C03576=1024.617,175.946,-114.492,168.623,47.960,159.009
C03577=1024.611,175.697,-114.469,168.619,47.965,159.010
C03578=1024.606,175.448,-114.447,168.616,47.970,159.010
C03579=1024.600,175.200,-114.424,168.612,47.974,159.011
C03580=1024.594,174.951,-114.401,168.609,47.979,159.011
C03581=1024.589,174.701,-114.379,168.605,47.983,159.011
C03582=1024.583,174.452,-114.356,168.602,47.988,159.012
C03583=1024.577,174.203,-114.335,168.598,47.993,159.012
C03584=1024.572,173.955,-114.312,168.594,47.997,159.013
C03585=1024.566,173.706,-114.289,168.591,48.002,159.013
C03586=1024.560,173.457,-114.268,168.587,48.006,159.014
C03587=1024.554,173.208,-114.245,168.584,48.011,159.014
C03588=1024.548,172.959,-114.222,168.580,48.016,159.015
C03589=1024.543,172.710,-114.200,168.576,48.020,159.015
C03590=1024.537,172.461,-114.178,168.573,48.025,159.015
C03591=1024.531,172.178,-114.152,168.570,48.030,159.016
C03592=1024.525,171.896,-114.126,168.565,48.035,159.016
C03593=1024.518,171.612,-114.102,168.562,48.040,159.017
C03594=1024.512,171.330,-114.076,168.558,48.046,159.018
C03595=1024.506,171.080,-114.054,168.554,48.051,159.018
C03596=1024.500,170.832,-114.031,168.550,48.055,159.018
C03597=1024.495,170.583,-114.010,168.547,48.059,159.019
C03598=1024.489,170.334,-113.987,168.544,48.064,159.019
C03599=1024.483,170.085,-113.965,168.541,48.069,159.020
C03600=1024.477,169.836,-113.942,168.537,48.073,159.020
C03601=1024.472,169.587,-113.920,168.534,48.078,159.021
C03602=1024.466,169.338,-113.899,168.530,48.082,159.021
C03603=1024.461,169.089,-113.876,168.527,48.087,159.022
C03604=1024.456,168.840,-113.854,168.523,48.091,159.022
C03605=1024.450,168.591,-113.831,168.519,48.096,159.022
C03606=1024.444,168.342,-113.809,168.517,48.101,159.023
C03607=1024.439,168.093,-113.787,168.513,48.105,159.023
C03608=1024.433,167.844,-113.764,168.510,48.110,159.024
C03609=1024.427,167.595,-113.743,168.506,48.114,159.024
C03610=1024.422,167.347,-113.720,168.503,48.119,159.025
C03611=1024.417,167.097,-113.698,168.499,48.124,159.025
C03612=1024.410,166.848,-113.676,168.497,48.128,159.026
C03613=1024.405,166.600,-113.654,168.493,48.132,159.026
C03614=1024.400,166.350,-113.631,168.489,48.137,159.026
C03615=1024.394,166.101,-113.610,168.486,48.142,159.027
C03616=1024.389,165.853,-113.587,168.483,48.147,159.027
C03617=1024.383,165.604,-113.565,168.479,48.152,159.028
C03618=1024.378,165.355,-113.544,168.476,48.155,159.028
C03619=1024.372,165.106,-113.522,168.473,48.160,159.029
C03620=1024.366,164.857,-113.499,168.469,48.165,159.029
C03621=1024.361,164.608,-113.477,168.466,48.170,159.030
C03622=1024.355,164.359,-113.455,168.462,48.174,159.030
C03623=1024.350,164.110,-113.433,168.460,48.178,159.031
C03624=1024.344,163.861,-113.411,168.456,48.183,159.031
C03625=1024.339,163.612,-113.389,168.453,48.188,159.032
C03626=1024.334,163.363,-113.367,168.449,48.192,159.032
C03627=1024.328,163.114,-113.345,168.446,48.197,159.032
C03628=1024.323,162.865,-113.323,168.443,48.201,159.033
C03629=1024.317,162.616,-113.300,168.439,48.206,159.033
C03630=1024.312,162.367,-113.279,168.436,48.211,159.034
C03631=1024.306,162.118,-113.257,168.433,48.215,159.034
C03632=1024.301,161.869,-113.235,168.430,48.220,159.035
C03633=1024.295,161.621,-113.213,168.426,48.224,159.035
C03634=1024.290,161.372,-113.191,168.423,48.229,159.036
C03635=1024.285,161.122,-113.169,168.420,48.233,159.036
C03636=1024.279,160.874,-113.147,168.417,48.238,159.037
C03637=1024.274,160.624,-113.125,168.413,48.243,159.037
C03638=1024.269,160.375,-113.103,168.410,48.247,159.037
C03639=1024.263,160.126,-113.082,168.407,48.251,159.038
C03640=1024.258,159.878,-113.059,168.403,48.256,159.038
C03641=1024.252,159.628,-113.037,168.400,48.261,159.039
C03642=1024.247,159.380,-113.015,168.397,48.265,159.039
C03643=1024.241,159.130,-112.993,168.394,48.270,159.040
C03644=1024.236,158.882,-112.972,168.391,48.275,159.040
C03645=1024.229,158.633,-112.950,168.387,48.280,159.041
C03646=1024.225,158.383,-112.929,168.384,48.285,159.041
C03647=1024.219,158.134,-112.908,168.381,48.289,159.042
C03648=1024.213,157.886,-112.886,168.378,48.294,159.042
C03649=1024.207,157.636,-112.865,168.374,48.299,159.043
C03650=1024.202,157.388,-112.843,168.371,48.303,159.043
C03651=1024.196,157.138,-112.821,168.367,48.308,159.044
C03652=1024.190,156.890,-112.800,168.365,48.313,159.044
C03653=1024.185,156.640,-112.779,168.361,48.318,159.045
C03654=1024.179,156.392,-112.758,168.358,48.322,159.045
C03655=1024.173,156.108,-112.732,168.355,48.327,159.046
C03656=1024.166,155.825,-112.708,168.350,48.333,159.046
C03657=1024.160,155.541,-112.684,168.347,48.339,159.047
C03658=1024.153,155.258,-112.660,168.343,48.344,159.047
C03659=1024.148,155.010,-112.638,168.340,48.348,159.048
C03660=1024.142,154.760,-112.617,168.337,48.353,159.048
C03661=1024.137,154.511,-112.596,168.333,48.358,159.049
C03662=1024.131,154.262,-112.574,168.330,48.363,159.049
C03663=1024.125,154.013,-112.553,168.328,48.367,159.050
C03664=1024.119,153.764,-112.532,168.324,48.372,159.050
C03665=1024.114,153.515,-112.510,168.321,48.377,159.051
C03666=1024.109,153.266,-112.489,168.317,48.382,159.051
C03667=1024.103,153.016,-112.468,168.315,48.386,159.052
C03668=1024.098,152.768,-112.446,168.311,48.391,159.052
C03669=1024.091,152.519,-112.425,168.308,48.396,159.053
C03670=1024.086,152.270,-112.404,168.305,48.401,159.053
C03671=1024.080,152.020,-112.383,168.302,48.406,159.054
C03672=1024.074,151.772,-112.361,168.299,48.411,159.054
C03673=1024.069,151.523,-112.341,168.295,48.415,159.055
C03674=1024.063,151.274,-112.319,168.292,48.420,159.055
C03675=1024.058,151.024,-112.299,168.289,48.425,159.056
C03676=1024.052,150.775,-112.277,168.286,48.430,159.056
C03677=1024.046,150.527,-112.256,168.283,48.434,159.057
C03678=1024.041,150.278,-112.235,168.279,48.439,159.057
C03679=1024.035,150.028,-112.214,168.277,48.444,159.058
C03680=1024.029,149.779,-112.193,168.273,48.449,159.058
C03681=1024.024,149.531,-112.171,168.270,48.453,159.059
C03682=1024.019,149.281,-112.150,168.266,48.458,159.059
C03683=1024.013,149.032,-112.129,168.264,48.463,159.060
C03684=1024.008,148.783,-112.108,168.260,48.468,159.060
C03685=1024.002,148.534,-112.087,168.257,48.473,159.061
C03686=1023.996,148.285,-112.066,168.255,48.477,159.061
C03687=1023.991,148.036,-112.045,168.251,48.483,159.062
C03688=1023.985,147.786,-112.024,168.248,48.487,159.063
C03689=1023.979,147.538,-112.003,168.245,48.492,159.063
C03690=1023.974,147.289,-111.982,168.242,48.497,159.064
C03691=1023.967,147.040,-111.961,168.239,48.502,159.064
C03692=1023.962,146.791,-111.941,168.235,48.506,159.065
C03693=1023.957,146.542,-111.920,168.233,48.511,159.065
C03694=1023.951,146.292,-111.898,168.229,48.516,159.066
C03695=1023.945,146.043,-111.878,168.226,48.521,159.066
C03696=1023.940,145.795,-111.857,168.224,48.525,159.067
C03697=1023.934,145.545,-111.836,168.220,48.531,159.067
C03698=1023.929,145.296,-111.815,168.217,48.536,159.068
C03699=1023.922,145.048,-111.794,168.214,48.540,159.068
C03700=1023.917,144.799,-111.774,168.211,48.545,159.069
C03701=1023.911,144.549,-111.753,168.208,48.550,159.069
C03702=1023.906,144.300,-111.732,168.204,48.555,159.070
C03703=1023.900,144.051,-111.712,168.202,48.560,159.070
C03704=1023.894,143.802,-111.691,168.199,48.565,159.071
C03705=1023.889,143.552,-111.670,168.195,48.570,159.071
C03706=1023.883,143.303,-111.650,168.192,48.574,159.072
C03707=1023.878,143.055,-111.628,168.189,48.579,159.072
C03708=1023.871,142.805,-111.608,168.186,48.584,159.073
C03709=1023.866,142.556,-111.588,168.183,48.589,159.073
C03710=1023.861,142.307,-111.567,168.181,48.594,159.074
C03711=1023.855,142.059,-111.546,168.177,48.599,159.074
C03712=1023.848,141.809,-111.525,168.174,48.604,159.075
C03713=1023.843,141.560,-111.505,168.171,48.608,159.076
C03714=1023.838,141.311,-111.484,168.168,48.613,159.076
C03715=1023.833,141.062,-111.464,168.164,48.618,159.076
C03716=1023.826,140.813,-111.443,168.162,48.623,159.077
C03717=1023.821,140.564,-111.422,168.159,48.628,159.078
C03718=1023.815,140.315,-111.402,168.155,48.633,159.078
C03719=1023.809,140.031,-111.378,168.152,48.638,159.079
C03720=1023.802,139.748,-111.355,168.149,48.644,159.079
C03721=1023.796,139.463,-111.332,168.145,48.649,159.080
C03722=1023.790,139.180,-111.308,168.142,48.655,159.080
C03723=1023.785,138.931,-111.287,168.139,48.659,159.081
C03724=1023.779,138.682,-111.267,168.136,48.664,159.081
C03725=1023.773,138.433,-111.247,168.133,48.670,159.082
C03726=1023.768,138.184,-111.226,168.130,48.674,159.083
C03727=1023.762,137.934,-111.205,168.127,48.679,159.083
C03728=1023.756,137.686,-111.185,168.123,48.684,159.084
C03729=1023.751,137.437,-111.164,168.121,48.688,159.084
C03730=1023.745,137.188,-111.144,168.118,48.694,159.085
C03731=1023.739,136.939,-111.124,168.115,48.699,159.085
C03732=1023.733,136.690,-111.104,168.112,48.703,159.086
C03733=1023.728,136.440,-111.083,168.109,48.708,159.086
C03734=1023.723,136.190,-111.063,168.106,48.714,159.087
C03735=1023.717,135.942,-111.043,168.103,48.718,159.087
C03736=1023.711,135.693,-111.022,168.100,48.723,159.088
C03737=1023.705,135.444,-111.002,168.096,48.728,159.088
C03738=1023.700,135.195,-110.982,168.094,48.733,159.089
C03739=1023.694,134.946,-110.962,168.091,48.738,159.090
C03740=1023.688,134.696,-110.941,168.087,48.743,159.090
C03741=1023.682,134.447,-110.921,168.085,48.748,159.091
C03742=1023.677,134.198,-110.901,168.082,48.753,159.091
C03743=1023.671,133.949,-110.881,168.079,48.758,159.092
C03744=1023.666,133.700,-110.860,168.076,48.763,159.092
C03745=1023.660,133.451,-110.841,168.073,48.768,159.093
C03746=1023.655,133.202,-110.820,168.070,48.772,159.093
C03747=1023.649,132.953,-110.800,168.067,48.778,159.094
C03748=1023.644,132.704,-110.780,168.064,48.783,159.094
C03749=1023.638,132.455,-110.760,168.061,48.787,159.095
C03750=1023.632,132.205,-110.739,168.058,48.792,159.095
C03751=1023.626,131.956,-110.719,168.055,48.797,159.096
C03752=1023.621,131.706,-110.699,168.053,48.802,159.097
C03753=1023.615,131.458,-110.679,168.049,48.807,159.097
C03754=1023.609,131.208,-110.659,168.047,48.812,159.098
C03755=1023.603,130.960,-110.639,168.043,48.817,159.098
C03756=1023.598,130.711,-110.618,168.040,48.822,159.099
C03757=1023.593,130.461,-110.599,168.038,48.827,159.099
C03758=1023.587,130.212,-110.579,168.034,48.832,159.100
C03759=1023.581,129.963,-110.558,168.032,48.836,159.100
C03760=1023.576,129.714,-110.539,168.029,48.842,159.101
C03761=1023.570,129.465,-110.519,168.026,48.847,159.101
C03762=1023.564,129.216,-110.499,168.023,48.851,159.102
C03763=1023.558,128.967,-110.480,168.020,48.857,159.103
C03764=1023.553,128.718,-110.459,168.017,48.862,159.103
C03765=1023.547,128.468,-110.440,168.015,48.867,159.104
C03766=1023.540,128.219,-110.420,168.011,48.872,159.104
C03767=1023.534,127.970,-110.400,168.008,48.877,159.105
C03768=1023.529,127.720,-110.381,168.006,48.882,159.105
C03769=1023.523,127.472,-110.361,168.002,48.887,159.106
C03770=1023.517,127.222,-110.341,167.999,48.892,159.106
C03771=1023.512,126.973,-110.321,167.997,48.897,159.107
C03772=1023.506,126.724,-110.302,167.994,48.902,159.108
C03773=1023.500,126.475,-110.282,167.990,48.908,159.108
C03774=1023.494,126.225,-110.262,167.988,48.912,159.109
C03775=1023.488,125.976,-110.242,167.985,48.917,159.109
C03776=1023.483,125.727,-110.223,167.982,48.923,159.110
C03777=1023.477,125.478,-110.203,167.979,48.927,159.110
C03778=1023.471,125.229,-110.183,167.976,48.932,159.111
C03779=1023.466,124.980,-110.163,167.974,48.938,159.112
C03780=1023.460,124.730,-110.144,167.970,48.942,159.112
C03781=1023.454,124.481,-110.124,167.967,48.947,159.113
C03782=1023.448,124.232,-110.105,167.965,48.953,159.113
C03783=1023.442,123.948,-110.083,167.961,48.958,159.114
C03784=1023.435,123.665,-110.060,167.958,48.964,159.114
C03785=1023.429,123.381,-110.038,167.955,48.970,159.115
C03786=1023.422,123.097,-110.016,167.952,48.975,159.116
C03787=1023.418,122.849,-109.995,167.948,48.980,159.116
C03788=1023.412,122.600,-109.976,167.946,48.985,159.117
C03789=1023.406,122.351,-109.956,167.943,48.990,159.117
C03790=1023.400,122.101,-109.937,167.939,48.995,159.118
C03791=1023.394,121.852,-109.917,167.937,49.001,159.119
C03792=1023.389,121.603,-109.898,167.934,49.005,159.119
C03793=1023.383,121.354,-109.879,167.932,49.010,159.120
C03794=1023.377,121.105,-109.859,167.928,49.015,159.120
C03795=1023.372,120.855,-109.839,167.926,49.020,159.121
C03796=1023.366,120.606,-109.820,167.923,49.025,159.121
C03797=1023.360,120.357,-109.800,167.919,49.030,159.122
C03798=1023.355,120.107,-109.780,167.917,49.035,159.122
C03799=1023.349,119.859,-109.761,167.914,49.040,159.123
C03800=1023.343,119.610,-109.741,167.912,49.045,159.123
C03801=1023.338,119.360,-109.722,167.909,49.051,159.124
C03802=1023.332,119.112,-109.702,167.906,49.055,159.125
C03803=1023.327,118.862,-109.682,167.903,49.060,159.125
C03804=1023.321,118.612,-109.663,167.900,49.065,159.126
C03805=1023.315,118.364,-109.643,167.897,49.070,159.126
C03806=1023.309,118.114,-109.624,167.894,49.075,159.127
C03807=1023.304,117.865,-109.605,167.892,49.080,159.127
C03808=1023.299,117.616,-109.586,167.888,49.085,159.128
C03809=1023.293,117.367,-109.566,167.886,49.090,159.128
C03810=1023.287,117.118,-109.547,167.883,49.095,159.129
C03811=1023.281,116.868,-109.527,167.881,49.100,159.130
C03812=1023.276,116.619,-109.507,167.877,49.104,159.130
C03813=1023.271,116.370,-109.488,167.875,49.110,159.131
C03814=1023.265,116.121,-109.469,167.872,49.115,159.131
C03815=1023.260,115.872,-109.450,167.869,49.119,159.132
C03816=1023.254,115.623,-109.430,167.866,49.124,159.132
C03817=1023.248,115.373,-109.410,167.864,49.130,159.133
C03818=1023.243,115.125,-109.391,167.861,49.135,159.133
C03819=1023.237,114.875,-109.372,167.858,49.139,159.134
C03820=1023.231,114.626,-109.353,167.855,49.144,159.134
C03821=1023.226,114.377,-109.332,167.853,49.149,159.135
C03822=1023.220,114.127,-109.313,167.849,49.154,159.136
C03823=1023.215,113.878,-109.294,167.847,49.159,159.136
C03824=1023.210,113.629,-109.275,167.844,49.164,159.137
C03825=1023.204,113.380,-109.256,167.841,49.168,159.137
C03826=1023.198,113.131,-109.236,167.838,49.174,159.138
C03827=1023.193,112.882,-109.217,167.836,49.179,159.138
C03828=1023.187,112.633,-109.198,167.833,49.184,159.139
C03829=1023.182,112.383,-109.178,167.830,49.188,159.139
C03830=1023.176,112.134,-109.159,167.827,49.194,159.140
C03831=1023.170,111.884,-109.140,167.825,49.199,159.140
C03832=1023.165,111.636,-109.121,167.821,49.203,159.141
C03833=1023.159,111.386,-109.102,167.819,49.209,159.142
C03834=1023.153,111.137,-109.083,167.816,49.214,159.142
C03835=1023.147,110.888,-109.064,167.814,49.219,159.143
C03836=1023.142,110.639,-109.045,167.811,49.224,159.143
C03837=1023.137,110.389,-109.026,167.808,49.229,159.144
C03838=1023.131,110.140,-109.007,167.805,49.234,159.144
C03839=1023.124,109.891,-108.988,167.802,49.239,159.145
C03840=1023.119,109.642,-108.969,167.800,49.244,159.145
C03841=1023.114,109.393,-108.950,167.797,49.249,159.146
C03842=1023.107,109.144,-108.931,167.794,49.254,159.147
C03843=1023.102,108.894,-108.912,167.791,49.260,159.147
C03844=1023.097,108.645,-108.894,167.789,49.264,159.148
C03845=1023.090,108.396,-108.875,167.785,49.269,159.148
C03846=1023.085,108.146,-108.856,167.783,49.275,159.149
C03847=1023.078,107.862,-108.834,167.779,49.281,159.150
C03848=1023.072,107.579,-108.813,167.776,49.286,159.150
C03849=1023.065,107.295,-108.791,167.773,49.292,159.151
C03850=1023.058,107.011,-108.770,167.770,49.298,159.151
C03851=1023.053,106.762,-108.751,167.767,49.303,159.152
C03852=1023.047,106.513,-108.733,167.765,49.308,159.153
C03853=1023.041,106.264,-108.714,167.762,49.313,159.153
C03854=1023.036,106.014,-108.694,167.760,49.318,159.154
C03855=1023.030,105.765,-108.677,167.756,49.323,159.154
C03856=1023.024,105.516,-108.657,167.754,49.328,159.155
C03857=1023.018,105.267,-108.639,167.751,49.333,159.155
C03858=1023.013,105.018,-108.620,167.749,49.339,159.156
C03859=1023.008,104.768,-108.601,167.746,49.344,159.157
C03860=1023.001,104.519,-108.583,167.743,49.348,159.157
C03861=1022.996,104.270,-108.564,167.740,49.354,159.158
C03862=1022.990,104.021,-108.545,167.738,49.359,159.158
C03863=1022.984,103.771,-108.527,167.734,49.364,159.159
C03864=1022.979,103.522,-108.508,167.731,49.369,159.159
C03865=1022.973,103.273,-108.489,167.729,49.374,159.160
C03866=1022.967,103.024,-108.470,167.726,49.379,159.160
C03867=1022.962,102.774,-108.452,167.724,49.384,159.161
C03868=1022.956,102.525,-108.433,167.721,49.389,159.162
C03869=1022.950,102.276,-108.414,167.718,49.394,159.162
C03870=1022.945,102.027,-108.395,167.716,49.399,159.163
C03871=1022.939,101.777,-108.377,167.713,49.404,159.163
C03872=1022.934,101.529,-108.358,167.710,49.409,159.164
C03873=1022.927,101.279,-108.340,167.707,49.414,159.165
C03874=1022.922,101.029,-108.321,167.705,49.419,159.165
C03875=1022.917,100.781,-108.302,167.702,49.424,159.166
C03876=1022.910,100.532,-108.283,167.700,49.429,159.166
C03877=1022.906,100.282,-108.265,167.696,49.434,159.167
C03878=1022.900,100.033,-108.246,167.694,49.439,159.167
C03879=1022.894,99.783,-108.228,167.691,49.445,159.168
C03880=1022.889,99.534,-108.209,167.689,49.449,159.168
C03881=1022.882,99.285,-108.191,167.685,49.454,159.169
C03882=1022.877,99.035,-108.172,167.683,49.460,159.170
C03883=1022.871,98.787,-108.154,167.680,49.465,159.170
C03884=1022.865,98.537,-108.136,167.678,49.470,159.171
C03885=1022.860,98.288,-108.117,167.675,49.475,159.171
C03886=1022.854,98.039,-108.099,167.673,49.480,159.172
C03887=1022.847,97.789,-108.080,167.669,49.485,159.172
C03888=1022.843,97.540,-108.062,167.666,49.490,159.173
C03889=1022.836,97.291,-108.044,167.664,49.496,159.174
C03890=1022.831,97.042,-108.026,167.661,49.501,159.174
C03891=1022.825,96.792,-108.008,167.659,49.506,159.175
C03892=1022.819,96.543,-107.989,167.655,49.511,159.175
C03893=1022.813,96.294,-107.971,167.653,49.516,159.176
C03894=1022.808,96.044,-107.952,167.650,49.521,159.176
C03895=1022.802,95.795,-107.934,167.648,49.526,159.177
C03896=1022.796,95.546,-107.916,167.645,49.532,159.178
C03897=1022.791,95.297,-107.898,167.642,49.536,159.178
C03898=1022.785,95.047,-107.880,167.639,49.542,159.179
C03899=1022.779,94.799,-107.861,167.637,49.547,159.179
C03900=1022.774,94.548,-107.843,167.634,49.552,159.180
C03901=1022.768,94.300,-107.825,167.632,49.557,159.181
C03902=1022.762,94.050,-107.807,167.628,49.562,159.181
C03903=1022.756,93.801,-107.789,167.626,49.567,159.182
C03904=1022.750,93.552,-107.770,167.623,49.572,159.182
C03905=1022.745,93.303,-107.752,167.621,49.577,159.183
C03906=1022.739,93.053,-107.734,167.618,49.583,159.183
C03907=1022.734,92.804,-107.716,167.616,49.587,159.184
C03908=1022.728,92.555,-107.698,167.612,49.592,159.184
C03909=1022.722,92.306,-107.679,167.610,49.598,159.185
C03910=1022.716,92.056,-107.661,167.607,49.603,159.185
C03911=1022.710,91.773,-107.640,167.604,49.608,159.186
C03912=1022.703,91.488,-107.620,167.601,49.614,159.187
C03913=1022.697,91.205,-107.599,167.598,49.620,159.187
C03914=1022.691,90.922,-107.579,167.595,49.625,159.188
C03915=1022.684,90.672,-107.561,167.593,49.631,159.189
C03916=1022.679,90.423,-107.542,167.590,49.636,159.189
C03917=1022.673,90.174,-107.524,167.587,49.640,159.190
C03918=1022.668,89.925,-107.506,167.584,49.646,159.190
C03919=1022.662,89.674,-107.488,167.582,49.651,159.191
C03920=1022.657,89.426,-107.469,167.579,49.656,159.191
C03921=1022.651,89.177,-107.452,167.577,49.661,159.192
C03922=1022.645,88.927,-107.434,167.573,49.666,159.193
C03923=1022.639,88.678,-107.416,167.571,49.672,159.193
C03924=1022.633,88.428,-107.398,167.568,49.677,159.194
C03925=1022.628,88.179,-107.381,167.566,49.682,159.194
C03926=1022.622,87.930,-107.363,167.563,49.687,159.195
C03927=1022.616,87.681,-107.345,167.561,49.692,159.196
C03928=1022.610,87.432,-107.327,167.558,49.697,159.196
C03929=1022.604,87.183,-107.309,167.555,49.702,159.197
C03930=1022.598,86.933,-107.291,167.552,49.708,159.197
C03931=1022.593,86.684,-107.274,167.550,49.712,159.198
C03932=1022.587,86.435,-107.256,167.547,49.718,159.198
C03933=1022.581,86.185,-107.238,167.545,49.723,159.199
C03934=1022.575,85.936,-107.221,167.542,49.728,159.200
C03935=1022.569,85.686,-107.203,167.539,49.733,159.200
C03936=1022.564,85.437,-107.185,167.536,49.739,159.201
C03937=1022.558,85.187,-107.167,167.534,49.744,159.201
C03938=1022.552,84.938,-107.150,167.531,49.749,159.202
C03939=1022.547,84.689,-107.132,167.529,49.754,159.202
C03940=1022.540,84.440,-107.114,167.526,49.759,159.203
C03941=1022.535,84.191,-107.097,167.524,49.764,159.204
C03942=1022.529,83.941,-107.079,167.520,49.769,159.204
C03943=1022.523,83.692,-107.061,167.518,49.774,159.205
C03944=1022.518,83.443,-107.043,167.515,49.780,159.205
C03945=1022.512,83.193,-107.026,167.513,49.784,159.206
C03946=1022.506,82.944,-107.008,167.510,49.790,159.206
C03947=1022.501,82.695,-106.990,167.508,49.795,159.207
C03948=1022.495,82.445,-106.972,167.504,49.800,159.207
C03949=1022.489,82.196,-106.955,167.502,49.805,159.208
C03950=1022.483,81.947,-106.937,167.499,49.810,159.209
C03951=1022.477,81.697,-106.919,167.497,49.816,159.209
C03952=1022.472,81.448,-106.902,167.494,49.821,159.210
C03953=1022.466,81.199,-106.884,167.491,49.825,159.210
C03954=1022.460,80.950,-106.866,167.489,49.831,159.211
C03955=1022.455,80.700,-106.849,167.486,49.836,159.211
C03956=1022.449,80.451,-106.831,167.484,49.841,159.212
C03957=1022.443,80.202,-106.813,167.481,49.846,159.213
C03958=1022.438,79.952,-106.796,167.479,49.851,159.213
C03959=1022.432,79.703,-106.779,167.475,49.856,159.214
C03960=1022.426,79.453,-106.761,167.473,49.861,159.214
C03961=1022.421,79.204,-106.743,167.470,49.866,159.215
C03962=1022.415,78.955,-106.726,167.468,49.871,159.215
C03963=1022.409,78.705,-106.708,167.465,49.877,159.216
C03964=1022.404,78.456,-106.690,167.463,49.882,159.216
C03965=1022.398,78.207,-106.673,167.460,49.886,159.217
C03966=1022.392,77.958,-106.655,167.457,49.891,159.217
C03967=1022.387,77.708,-106.638,167.455,49.897,159.218
C03968=1022.381,77.459,-106.620,167.452,49.902,159.219
C03969=1022.376,77.210,-106.603,167.449,49.906,159.219
C03970=1022.369,76.960,-106.585,167.446,49.912,159.220
C03971=1022.364,76.711,-106.569,167.444,49.917,159.220
C03972=1022.358,76.462,-106.551,167.441,49.923,159.221
C03973=1022.353,76.213,-106.533,167.439,49.927,159.222
C03974=1022.346,75.963,-106.516,167.436,49.932,159.222
C03975=1022.340,75.679,-106.496,167.433,49.939,159.223
C03976=1022.333,75.396,-106.476,167.430,49.945,159.223
C03977=1022.327,75.112,-106.457,167.427,49.950,159.224
C03978=1022.320,74.828,-106.438,167.424,49.956,159.225
C03979=1022.314,74.579,-106.420,167.421,49.962,159.225
C03980=1022.309,74.330,-106.403,167.419,49.966,159.226
C03981=1022.302,74.080,-106.386,167.417,49.971,159.226
C03982=1022.297,73.831,-106.368,167.414,49.977,159.227
C03983=1022.292,73.582,-106.351,167.411,49.982,159.228
C03984=1022.285,73.333,-106.334,167.409,49.987,159.228
C03985=1022.279,73.083,-106.316,167.406,49.992,159.229
C03986=1022.274,72.833,-106.300,167.403,49.997,159.229
C03987=1022.268,72.584,-106.282,167.401,50.003,159.230
C03988=1022.262,72.335,-106.266,167.398,50.008,159.230
C03989=1022.256,72.085,-106.248,167.395,50.012,159.231
C03990=1022.251,71.836,-106.230,167.393,50.018,159.231
C03991=1022.245,71.587,-106.214,167.390,50.023,159.232
C03992=1022.239,71.338,-106.197,167.387,50.028,159.232
C03993=1022.234,71.088,-106.180,167.385,50.033,159.233
C03994=1022.227,70.839,-106.162,167.382,50.038,159.234
C03995=1022.222,70.589,-106.145,167.380,50.044,159.234
C03996=1022.217,70.340,-106.128,167.377,50.049,159.235
C03997=1022.211,70.091,-106.112,167.374,50.053,159.235
C03998=1022.205,69.842,-106.094,167.372,50.059,159.236
C03999=1022.200,69.593,-106.077,167.369,50.064,159.236
C04000=1022.193,69.343,-106.060,167.367,50.069,159.237
C04001=1022.188,69.094,-106.042,167.364,50.074,159.238
C04002=1022.182,68.844,-106.025,167.362,50.079,159.238
C04003=1022.176,68.595,-106.008,167.358,50.084,159.239
C04004=1022.171,68.346,-105.992,167.356,50.090,159.239
C04005=1022.164,68.095,-105.975,167.353,50.095,159.240
C04006=1022.159,67.846,-105.957,167.351,50.099,159.240
C04007=1022.153,67.597,-105.941,167.348,50.105,159.241
C04008=1022.147,67.348,-105.924,167.346,50.110,159.242
C04009=1022.141,67.099,-105.907,167.343,50.116,159.242
C04010=1022.136,66.850,-105.890,167.340,50.120,159.243
C04011=1022.130,66.600,-105.874,167.337,50.125,159.243
C04012=1022.124,66.350,-105.856,167.335,50.131,159.244
C04013=1022.118,66.101,-105.839,167.332,50.136,159.244
C04014=1022.113,65.852,-105.823,167.330,50.141,159.245
C04015=1022.107,65.602,-105.806,167.327,50.146,159.245
C04016=1022.101,65.353,-105.789,167.325,50.151,159.246
C04017=1022.095,65.104,-105.772,167.323,50.157,159.247
C04018=1022.090,64.854,-105.756,167.319,50.162,159.247
C04019=1022.084,64.605,-105.739,167.317,50.166,159.248
C04020=1022.078,64.355,-105.721,167.314,50.172,159.248
C04021=1022.072,64.106,-105.705,167.312,50.177,159.249
C04022=1022.066,63.857,-105.688,167.309,50.182,159.249
C04023=1022.060,63.607,-105.671,167.307,50.187,159.250
C04024=1022.055,63.358,-105.654,167.303,50.193,159.250
C04025=1022.049,63.108,-105.638,167.301,50.197,159.251
C04026=1022.043,62.860,-105.621,167.298,50.203,159.252
C04027=1022.037,62.610,-105.605,167.296,50.208,159.252
C04028=1022.031,62.360,-105.588,167.293,50.214,159.253
C04029=1022.025,62.111,-105.571,167.291,50.218,159.253
C04030=1022.019,61.861,-105.555,167.288,50.224,159.254
C04031=1022.013,61.612,-105.539,167.285,50.229,159.254
C04032=1022.007,61.362,-105.523,167.283,50.235,159.255
C04033=1022.001,61.114,-105.506,167.280,50.240,159.256
C04034=1021.996,60.864,-105.489,167.278,50.245,159.256
C04035=1021.990,60.615,-105.473,167.274,50.250,159.257
C04036=1021.984,60.365,-105.456,167.273,50.256,159.257
C04037=1021.978,60.116,-105.440,167.269,50.261,159.258
C04038=1021.972,59.867,-105.424,167.267,50.266,159.259
C04039=1021.965,59.549,-105.403,167.264,50.273,159.259
C04040=1021.957,59.232,-105.382,167.260,50.280,159.260
C04041=1021.950,58.915,-105.362,167.257,50.287,159.261
C04042=1021.942,58.598,-105.340,167.254,50.293,159.262
C04043=1021.937,58.348,-105.323,167.251,50.298,159.262
C04044=1021.931,58.099,-105.307,167.248,50.304,159.263
C04045=1021.924,57.849,-105.290,167.246,50.309,159.263
C04046=1021.918,57.599,-105.274,167.242,50.314,159.264
C04047=1021.912,57.350,-105.258,167.241,50.319,159.264
C04048=1021.906,57.101,-105.242,167.237,50.324,159.265
C04049=1021.900,56.851,-105.225,167.235,50.330,159.265
C04050=1021.895,56.602,-105.209,167.232,50.335,159.266
C04051=1021.889,56.352,-105.192,167.230,50.340,159.266
C04052=1021.883,56.103,-105.176,167.227,50.345,159.267
C04053=1021.877,55.854,-105.160,167.225,50.350,159.268
C04054=1021.871,55.604,-105.144,167.222,50.356,159.268
C04055=1021.865,55.355,-105.127,167.220,50.361,159.269
C04056=1021.859,55.106,-105.111,167.216,50.366,159.269
C04057=1021.854,54.856,-105.094,167.215,50.371,159.270
C04058=1021.848,54.607,-105.078,167.211,50.376,159.270
C04059=1021.843,54.358,-105.062,167.209,50.381,159.271
C04060=1021.837,54.109,-105.046,167.206,50.387,159.271
C04061=1021.831,53.859,-105.030,167.204,50.392,159.272
C04062=1021.825,53.609,-105.014,167.201,50.397,159.273
C04063=1021.819,53.360,-104.998,167.199,50.402,159.273
C04064=1021.813,53.111,-104.981,167.196,50.407,159.274
C04065=1021.808,52.861,-104.965,167.194,50.413,159.274
C04066=1021.802,52.612,-104.948,167.190,50.418,159.275
C04067=1021.796,52.362,-104.932,167.188,50.423,159.275
C04068=1021.790,52.113,-104.916,167.185,50.428,159.276
C04069=1021.784,51.864,-104.900,167.183,50.433,159.276
C04070=1021.778,51.614,-104.883,167.180,50.438,159.277
C04071=1021.774,51.381,-104.868,167.178,50.443,159.277
C04072=1021.768,51.149,-104.853,167.175,50.448,159.278
C04073=1021.763,50.916,-104.838,167.173,50.453,159.278
C04074=1021.757,50.684,-104.823,167.171,50.457,159.279
C04075=1021.752,50.450,-104.808,167.169,50.462,159.280
C04076=1021.747,50.218,-104.793,167.165,50.467,159.280
C04077=1021.742,49.985,-104.778,167.163,50.472,159.280
C04078=1021.736,49.752,-104.763,167.161,50.476,159.281
C04079=1021.730,49.503,-104.747,167.159,50.482,159.282
C04080=1021.725,49.254,-104.731,167.155,50.487,159.282
C04081=1021.719,49.005,-104.714,167.153,50.492,159.283
C04082=1021.713,48.756,-104.698,167.150,50.497,159.283
C04083=1021.708,48.505,-104.682,167.148,50.502,159.284
C04084=1021.702,48.256,-104.666,167.145,50.507,159.284
C04085=1021.696,48.007,-104.650,167.143,50.512,159.285
C04086=1021.690,47.757,-104.633,167.140,50.517,159.285
C04087=1021.684,47.509,-104.617,167.137,50.523,159.286
C04088=1021.679,47.259,-104.602,167.135,50.527,159.286
C04089=1021.673,47.009,-104.586,167.132,50.533,159.287
C04090=1021.667,46.760,-104.569,167.130,50.537,159.287
C04091=1021.661,46.511,-104.553,167.127,50.542,159.288
C04092=1021.656,46.260,-104.537,167.125,50.548,159.288
C04093=1021.651,46.012,-104.521,167.122,50.553,159.289
C04094=1021.645,45.762,-104.505,167.119,50.558,159.289
C04095=1021.639,45.513,-104.489,167.117,50.563,159.290
C04096=1021.633,45.263,-104.473,167.114,50.568,159.290
C04097=1021.627,45.014,-104.457,167.112,50.572,159.291
C04098=1021.622,44.765,-104.441,167.109,50.578,159.292
C04099=1021.616,44.516,-104.425,167.106,50.583,159.292
C04100=1021.610,44.266,-104.409,167.104,50.588,159.293
C04101=1021.604,44.016,-104.393,167.101,50.593,159.293
C04102=1021.599,43.767,-104.376,167.099,50.598,159.294
C04103=1021.593,43.483,-104.359,167.096,50.604,159.294
C04104=1021.586,43.199,-104.340,167.093,50.609,159.295
C04105=1021.580,42.914,-104.322,167.090,50.615,159.295
C04106=1021.574,42.631,-104.304,167.087,50.620,159.296
C04107=1021.568,42.382,-104.287,167.084,50.626,159.296
C04108=1021.562,42.132,-104.272,167.082,50.631,159.297
C04109=1021.556,41.883,-104.256,167.079,50.636,159.297
C04110=1021.551,41.633,-104.241,167.076,50.641,159.298
C04111=1021.545,41.384,-104.225,167.074,50.647,159.299
C04112=1021.539,41.134,-104.209,167.071,50.652,159.299
C04113=1021.532,40.885,-104.193,167.068,50.657,159.299
C04114=1021.527,40.636,-104.178,167.066,50.661,159.300
C04115=1021.521,40.386,-104.162,167.063,50.667,159.301
C04116=1021.516,40.136,-104.146,167.061,50.672,159.301
C04117=1021.510,39.887,-104.130,167.058,50.677,159.302
C04118=1021.505,39.638,-104.115,167.055,50.682,159.302
C04119=1021.498,39.388,-104.100,167.052,50.688,159.303
C04120=1021.492,39.139,-104.084,167.050,50.693,159.303
C04121=1021.487,38.889,-104.068,167.047,50.698,159.304
C04122=1021.481,38.640,-104.052,167.045,50.703,159.304
C04123=1021.476,38.390,-104.037,167.042,50.708,159.305
C04124=1021.469,38.141,-104.021,167.040,50.713,159.305
C04125=1021.463,37.891,-104.006,167.038,50.718,159.306
C04126=1021.458,37.643,-103.990,167.034,50.723,159.306
C04127=1021.452,37.393,-103.974,167.032,50.728,159.307
C04128=1021.447,37.143,-103.959,167.029,50.733,159.307
C04129=1021.441,36.894,-103.943,167.027,50.739,159.308
C04130=1021.435,36.644,-103.928,167.024,50.744,159.308
C04131=1021.429,36.394,-103.912,167.022,50.749,159.309
C04132=1021.423,36.145,-103.897,167.018,50.754,159.309
C04133=1021.418,35.896,-103.881,167.017,50.759,159.310
C04134=1021.412,35.646,-103.866,167.013,50.764,159.311
C04135=1021.406,35.396,-103.851,167.011,50.769,159.311
C04136=1021.400,35.148,-103.835,167.008,50.775,159.312
C04137=1021.394,34.898,-103.820,167.006,50.780,159.312
C04138=1021.388,34.648,-103.805,167.003,50.785,159.313
C04139=1021.382,34.399,-103.790,167.000,50.790,159.313
C04140=1021.376,34.150,-103.774,166.998,50.796,159.314
C04141=1021.371,33.900,-103.758,166.995,50.801,159.314
C04142=1021.365,33.651,-103.744,166.992,50.806,159.315
C04143=1021.359,33.401,-103.728,166.990,50.811,159.315
C04144=1021.353,33.152,-103.712,166.987,50.816,159.316
C04145=1021.348,32.903,-103.697,166.984,50.821,159.316
C04146=1021.341,32.653,-103.682,166.982,50.826,159.317
C04147=1021.336,32.403,-103.667,166.979,50.831,159.317
C04148=1021.330,32.154,-103.652,166.977,50.837,159.318
C04149=1021.324,31.904,-103.637,166.974,50.842,159.318
C04150=1021.318,31.655,-103.620,166.972,50.847,159.319
C04151=1021.312,31.406,-103.606,166.968,50.852,159.319
C04152=1021.307,31.156,-103.590,166.966,50.858,159.320
C04153=1021.301,30.907,-103.576,166.963,50.863,159.320
C04154=1021.295,30.657,-103.560,166.961,50.867,159.321
C04155=1021.289,30.407,-103.545,166.958,50.873,159.321
C04156=1021.284,30.159,-103.529,166.956,50.877,159.322
C04157=1021.277,29.909,-103.514,166.953,50.883,159.323
C04158=1021.272,29.660,-103.499,166.951,50.888,159.323
C04159=1021.267,29.410,-103.484,166.947,50.893,159.324
C04160=1021.260,29.160,-103.469,166.945,50.898,159.324
C04161=1021.255,28.911,-103.454,166.942,50.903,159.324
C04162=1021.249,28.661,-103.439,166.940,50.908,159.325
C04163=1021.244,28.412,-103.423,166.937,50.913,159.325
C04164=1021.237,28.162,-103.408,166.935,50.919,159.326
C04165=1021.232,27.912,-103.393,166.932,50.924,159.327
C04166=1021.226,27.663,-103.378,166.929,50.929,159.327
C04167=1021.219,27.379,-103.361,166.927,50.935,159.328
C04168=1021.213,27.095,-103.344,166.924,50.941,159.328
C04169=1021.206,26.811,-103.327,166.920,50.947,159.329
C04170=1021.199,26.527,-103.310,166.917,50.953,159.329
C04171=1021.194,26.277,-103.295,166.915,50.957,159.330
C04172=1021.188,26.028,-103.280,166.912,50.963,159.330
C04173=1021.182,25.779,-103.265,166.909,50.967,159.331
C04174=1021.176,25.529,-103.250,166.906,50.973,159.331
C04175=1021.170,25.279,-103.235,166.904,50.978,159.332
C04176=1021.164,25.030,-103.220,166.901,50.983,159.332
C04177=1021.159,24.780,-103.205,166.899,50.988,159.333
C04178=1021.153,24.531,-103.190,166.896,50.993,159.333
C04179=1021.147,24.282,-103.175,166.893,50.999,159.334
C04180=1021.141,24.032,-103.160,166.891,51.004,159.335
C04181=1021.135,23.782,-103.146,166.888,51.009,159.335
C04182=1021.130,23.533,-103.131,166.885,51.014,159.335
C04183=1021.123,23.284,-103.116,166.882,51.019,159.336
C04184=1021.118,23.034,-103.101,166.881,51.025,159.337
C04185=1021.112,22.785,-103.086,166.877,51.030,159.337
C04186=1021.106,22.536,-103.071,166.875,51.035,159.338
C04187=1021.100,22.286,-103.056,166.872,51.040,159.338
C04188=1021.095,22.036,-103.042,166.870,51.045,159.339
C04189=1021.089,21.786,-103.027,166.867,51.050,159.339
C04190=1021.083,21.537,-103.012,166.864,51.055,159.339
C04191=1021.077,21.288,-102.997,166.862,51.061,159.340
C04192=1021.071,21.039,-102.982,166.859,51.065,159.341
C04193=1021.066,20.789,-102.968,166.856,51.071,159.341
C04194=1021.060,20.539,-102.953,166.854,51.076,159.342
C04195=1021.054,20.290,-102.938,166.851,51.081,159.342
C04196=1021.048,20.040,-102.923,166.849,51.086,159.342
C04197=1021.043,19.791,-102.908,166.845,51.091,159.343
C04198=1021.037,19.541,-102.894,166.843,51.096,159.343
C04199=1021.031,19.292,-102.879,166.840,51.101,159.344
C04200=1021.025,19.042,-102.864,166.837,51.107,159.344
C04201=1021.020,18.792,-102.850,166.835,51.111,159.345
C04202=1021.014,18.543,-102.835,166.832,51.117,159.345
C04203=1021.008,18.294,-102.820,166.830,51.122,159.346
C04204=1021.002,18.044,-102.807,166.827,51.127,159.346
C04205=1020.996,17.795,-102.792,166.825,51.132,159.347
C04206=1020.990,17.546,-102.777,166.822,51.137,159.347
C04207=1020.984,17.295,-102.763,166.819,51.142,159.348
C04208=1020.979,17.046,-102.748,166.816,51.147,159.348
C04209=1020.973,16.797,-102.733,166.814,51.152,159.349
C04210=1020.967,16.547,-102.719,166.811,51.158,159.349
C04211=1020.961,16.298,-102.704,166.808,51.163,159.350
C04212=1020.955,16.048,-102.689,166.805,51.168,159.350
C04213=1020.950,15.799,-102.675,166.803,51.173,159.351
C04214=1020.944,15.550,-102.661,166.801,51.178,159.351
C04215=1020.938,15.299,-102.646,166.797,51.183,159.352
C04216=1020.933,15.050,-102.631,166.795,51.188,159.352
C04217=1020.927,14.801,-102.618,166.792,51.194,159.353
C04218=1020.921,14.551,-102.603,166.790,51.198,159.353
C04219=1020.915,14.302,-102.588,166.787,51.204,159.354
C04220=1020.910,14.052,-102.574,166.784,51.208,159.354
C04221=1020.903,13.803,-102.559,166.781,51.214,159.355
C04222=1020.898,13.553,-102.545,166.779,51.219,159.355
C04223=1020.892,13.303,-102.530,166.776,51.224,159.356
C04224=1020.886,13.054,-102.517,166.773,51.230,159.356
C04225=1020.880,12.805,-102.502,166.771,51.234,159.357
C04226=1020.874,12.555,-102.488,166.768,51.240,159.357
C04227=1020.868,12.305,-102.474,166.766,51.245,159.358
C04228=1020.863,12.056,-102.459,166.763,51.250,159.358
C04229=1020.857,11.806,-102.445,166.760,51.256,159.359
C04230=1020.851,11.557,-102.431,166.757,51.261,159.359
C04231=1020.844,11.274,-102.415,166.755,51.266,159.360
C04232=1020.837,10.992,-102.399,166.751,51.273,159.360
C04233=1020.831,10.709,-102.383,166.748,51.279,159.361
C04234=1020.824,10.426,-102.367,166.745,51.284,159.361
C04235=1020.818,10.177,-102.353,166.742,51.290,159.362
C04236=1020.813,9.928,-102.339,166.740,51.295,159.362
C04237=1020.806,9.678,-102.325,166.737,51.300,159.363
C04238=1020.800,9.429,-102.311,166.734,51.305,159.363
C04239=1020.795,9.179,-102.297,166.731,51.310,159.364
C04240=1020.789,8.929,-102.282,166.729,51.316,159.364
C04241=1020.783,8.680,-102.268,166.727,51.321,159.365
C04242=1020.778,8.430,-102.254,166.723,51.326,159.365
C04243=1020.772,8.181,-102.240,166.720,51.331,159.366
C04244=1020.765,7.931,-102.226,166.718,51.336,159.366
C04245=1020.759,7.682,-102.212,166.715,51.341,159.367
C04246=1020.754,7.432,-102.198,166.713,51.346,159.367
C04247=1020.749,7.183,-102.184,166.710,51.351,159.368
C04248=1020.742,6.933,-102.169,166.707,51.356,159.368
C04249=1020.737,6.683,-102.155,166.705,51.362,159.369
C04250=1020.730,6.434,-102.142,166.701,51.367,159.369
C04251=1020.725,6.185,-102.128,166.699,51.372,159.370
C04252=1020.719,5.934,-102.114,166.696,51.377,159.370
C04253=1020.713,5.685,-102.099,166.694,51.382,159.371
C04254=1020.708,5.436,-102.086,166.691,51.387,159.371
C04255=1020.702,5.186,-102.072,166.688,51.393,159.371
C04256=1020.696,4.937,-102.058,166.685,51.398,159.372
C04257=1020.690,4.687,-102.043,166.682,51.403,159.372
C04258=1020.684,4.438,-102.030,166.680,51.408,159.373
C04259=1020.679,4.188,-102.016,166.677,51.413,159.373
C04260=1020.673,3.939,-102.002,166.675,51.418,159.374
C04261=1020.668,3.689,-101.988,166.672,51.423,159.374
C04262=1020.661,3.439,-101.974,166.670,51.428,159.375
C04263=1020.655,3.190,-101.960,166.666,51.433,159.375
C04264=1020.650,2.940,-101.946,166.663,51.438,159.375
C04265=1020.644,2.691,-101.932,166.661,51.443,159.376
C04266=1020.639,2.441,-101.918,166.658,51.448,159.376
C04267=1020.633,2.192,-101.904,166.656,51.453,159.377
C04268=1020.626,1.942,-101.891,166.653,51.458,159.377
C04269=1020.621,1.692,-101.877,166.650,51.463,159.378
C04270=1020.615,1.443,-101.863,166.647,51.469,159.378
C04271=1020.610,1.194,-101.848,166.645,51.473,159.379
C04272=1020.604,0.944,-101.835,166.642,51.479,159.379
C04273=1020.598,0.695,-101.821,166.639,51.484,159.380
C04274=1020.592,0.445,-101.807,166.637,51.489,159.380
C04275=1020.587,0.196,-101.794,166.634,51.494,159.380
C04276=1020.581,-0.055,-101.779,166.631,51.499,159.381
C04277=1020.575,-0.304,-101.765,166.628,51.504,159.381
C04278=1020.570,-0.554,-101.752,166.626,51.509,159.382
C04279=1020.564,-0.803,-101.738,166.623,51.514,159.382
C04280=1020.558,-1.053,-101.724,166.620,51.518,159.383
C04281=1020.553,-1.302,-101.711,166.617,51.524,159.383
C04282=1020.547,-1.552,-101.697,166.615,51.529,159.384
C04283=1020.542,-1.801,-101.683,166.612,51.534,159.384
C04284=1020.536,-2.051,-101.670,166.610,51.539,159.384
C04285=1020.530,-2.300,-101.656,166.607,51.544,159.385
C04286=1020.525,-2.550,-101.642,166.605,51.549,159.385
C04287=1020.519,-2.799,-101.628,166.601,51.553,159.386
C04288=1020.513,-3.050,-101.614,166.598,51.559,159.386
C04289=1020.507,-3.299,-101.601,166.596,51.564,159.387
C04290=1020.501,-3.548,-101.587,166.593,51.569,159.387
C04291=1020.496,-3.798,-101.573,166.590,51.574,159.387
C04292=1020.490,-4.048,-101.559,166.587,51.579,159.388
C04293=1020.485,-4.297,-101.545,166.585,51.584,159.388
C04294=1020.479,-4.546,-101.532,166.582,51.589,159.389
C04295=1020.473,-4.827,-101.517,166.579,51.594,159.389
C04296=1020.466,-5.108,-101.502,166.576,51.600,159.390
C04297=1020.459,-5.389,-101.487,166.573,51.606,159.390
C04298=1020.453,-5.670,-101.472,166.569,51.612,159.391
C04299=1020.447,-5.919,-101.459,166.567,51.617,159.391
C04300=1020.441,-6.168,-101.445,166.564,51.623,159.392
C04301=1020.435,-6.418,-101.432,166.561,51.628,159.392
C04302=1020.430,-6.668,-101.418,166.559,51.633,159.393
C04303=1020.423,-6.917,-101.405,166.556,51.638,159.393
C04304=1020.418,-7.167,-101.391,166.554,51.643,159.394
C04305=1020.412,-7.416,-101.378,166.551,51.648,159.394
C04306=1020.407,-7.666,-101.365,166.547,51.653,159.394
C04307=1020.400,-7.915,-101.352,166.545,51.658,159.395
C04308=1020.394,-8.165,-101.338,166.542,51.664,159.395
C04309=1020.389,-8.415,-101.325,166.539,51.669,159.396
C04310=1020.383,-8.664,-101.312,166.537,51.674,159.396
C04311=1020.377,-8.914,-101.298,166.533,51.678,159.396
C04312=1020.371,-9.164,-101.285,166.531,51.683,159.397
C04313=1020.366,-9.413,-101.272,166.528,51.688,159.397
C04314=1020.360,-9.662,-101.258,166.525,51.694,159.398
C04315=1020.355,-9.913,-101.245,166.523,51.699,159.398
C04316=1020.348,-10.162,-101.232,166.520,51.704,159.399
C04317=1020.342,-10.411,-101.219,166.517,51.709,159.399
C04318=1020.337,-10.661,-101.205,166.514,51.714,159.400
C04319=1020.331,-10.911,-101.192,166.511,51.719,159.400
C04320=1020.326,-11.160,-101.179,166.509,51.724,159.400
C04321=1020.320,-11.409,-101.166,166.506,51.730,159.401
C04322=1020.314,-11.659,-101.152,166.503,51.735,159.401
C04323=1020.309,-11.909,-101.140,166.501,51.740,159.402
C04324=1020.302,-12.158,-101.126,166.498,51.745,159.402
C04325=1020.297,-12.408,-101.113,166.495,51.749,159.402
C04326=1020.291,-12.658,-101.100,166.492,51.754,159.403
C04327=1020.285,-12.907,-101.086,166.489,51.760,159.403
C04328=1020.280,-13.157,-101.074,166.487,51.765,159.404
C04329=1020.274,-13.407,-101.060,166.484,51.770,159.404
C04330=1020.269,-13.656,-101.048,166.481,51.775,159.405
C04331=1020.263,-13.905,-101.034,166.478,51.780,159.405
C04332=1020.257,-14.155,-101.021,166.476,51.784,159.405
C04333=1020.251,-14.405,-101.008,166.473,51.790,159.406
C04334=1020.246,-14.655,-100.995,166.470,51.795,159.406
C04335=1020.240,-14.904,-100.981,166.467,51.800,159.407
C04336=1020.234,-15.154,-100.969,166.464,51.805,159.407
C04337=1020.229,-15.403,-100.955,166.462,51.809,159.407
C04338=1020.223,-15.653,-100.943,166.459,51.814,159.408
C04339=1020.218,-15.902,-100.929,166.456,51.820,159.408
C04340=1020.212,-16.152,-100.916,166.453,51.825,159.409
C04341=1020.206,-16.401,-100.903,166.450,51.830,159.409
C04342=1020.200,-16.651,-100.891,166.447,51.835,159.409
C04343=1020.194,-16.901,-100.878,166.445,51.840,159.410
C04344=1020.189,-17.150,-100.865,166.442,51.845,159.410
C04345=1020.183,-17.400,-100.852,166.439,51.851,159.411
C04346=1020.177,-17.650,-100.839,166.437,51.856,159.411
C04347=1020.171,-17.899,-100.826,166.434,51.861,159.412
C04348=1020.165,-18.149,-100.814,166.430,51.866,159.412
C04349=1020.160,-18.398,-100.801,166.428,51.871,159.413
C04350=1020.153,-18.647,-100.788,166.425,51.876,159.413
C04351=1020.148,-18.898,-100.775,166.422,51.881,159.413
C04352=1020.142,-19.147,-100.763,166.420,51.886,159.414
C04353=1020.136,-19.397,-100.750,166.416,51.891,159.414
C04354=1020.131,-19.646,-100.737,166.413,51.896,159.414
C04355=1020.125,-19.896,-100.724,166.411,51.901,159.415
C04356=1020.119,-20.146,-100.712,166.408,51.907,159.415
C04357=1020.113,-20.396,-100.699,166.406,51.912,159.416
C04358=1020.108,-20.644,-100.686,166.403,51.917,159.416
C04359=1020.101,-20.923,-100.672,166.400,51.922,159.417
C04360=1020.094,-21.203,-100.658,166.397,51.928,159.417
C04361=1020.089,-21.481,-100.644,166.393,51.934,159.418
C04362=1020.082,-21.761,-100.629,166.390,51.939,159.418
C04363=1020.077,-22.010,-100.617,166.388,51.944,159.418
C04364=1020.071,-22.259,-100.604,166.384,51.949,159.419
C04365=1020.065,-22.509,-100.591,166.381,51.955,159.419
C04366=1020.059,-22.758,-100.579,166.379,51.959,159.420
C04367=1020.053,-23.008,-100.566,166.376,51.965,159.420
C04368=1020.048,-23.258,-100.554,166.373,51.969,159.420
C04369=1020.042,-23.508,-100.541,166.371,51.974,159.421
C04370=1020.037,-23.757,-100.528,166.367,51.980,159.421
C04371=1020.031,-24.007,-100.515,166.364,51.985,159.422
C04372=1020.025,-24.257,-100.503,166.362,51.989,159.422
C04373=1020.020,-24.506,-100.491,166.359,51.994,159.422
C04374=1020.014,-24.756,-100.478,166.357,51.999,159.423
C04375=1020.008,-25.006,-100.465,166.353,52.005,159.423
C04376=1020.003,-25.255,-100.453,166.350,52.010,159.424
C04377=1019.997,-25.505,-100.440,166.348,52.014,159.424
C04378=1019.991,-25.755,-100.428,166.345,52.019,159.424
C04379=1019.986,-26.003,-100.415,166.343,52.024,159.425
C04380=1019.980,-26.253,-100.402,166.340,52.030,159.425
C04381=1019.974,-26.503,-100.390,166.336,52.034,159.425
C04382=1019.969,-26.752,-100.377,166.334,52.039,159.426
C04383=1019.963,-27.002,-100.365,166.331,52.045,159.426
C04384=1019.957,-27.252,-100.352,166.327,52.049,159.426
C04385=1019.952,-27.502,-100.339,166.325,52.054,159.427
C04386=1019.946,-27.752,-100.327,166.322,52.059,159.427
C04387=1019.940,-28.001,-100.315,166.320,52.064,159.428
C04388=1019.934,-28.250,-100.303,166.317,52.070,159.428
C04389=1019.929,-28.501,-100.291,166.314,52.075,159.429
C04390=1019.924,-28.750,-100.279,166.310,52.079,159.429
C04391=1019.918,-29.000,-100.266,166.308,52.084,159.429
C04392=1019.912,-29.250,-100.254,166.305,52.090,159.430
C04393=1019.906,-29.499,-100.241,166.302,52.095,159.430
C04394=1019.900,-29.748,-100.229,166.300,52.100,159.431
C04395=1019.895,-29.998,-100.217,166.297,52.105,159.431
C04396=1019.889,-30.248,-100.205,166.294,52.111,159.431
C04397=1019.883,-30.498,-100.193,166.291,52.115,159.432
C04398=1019.878,-30.747,-100.181,166.288,52.120,159.432
C04399=1019.872,-30.997,-100.168,166.285,52.125,159.432
C04400=1019.866,-31.246,-100.157,166.282,52.131,159.433
C04401=1019.860,-31.496,-100.144,166.280,52.136,159.433
C04402=1019.855,-31.745,-100.132,166.276,52.140,159.433
C04403=1019.849,-31.996,-100.120,166.273,52.146,159.434
C04404=1019.843,-32.245,-100.107,166.271,52.151,159.434
C04405=1019.838,-32.495,-100.095,166.268,52.156,159.435
C04406=1019.831,-32.744,-100.083,166.265,52.161,159.435
C04407=1019.826,-32.994,-100.072,166.262,52.165,159.435
C04408=1019.820,-33.244,-100.059,166.259,52.171,159.436
C04409=1019.815,-33.493,-100.047,166.256,52.176,159.436
C04410=1019.809,-33.743,-100.035,166.254,52.181,159.437
C04411=1019.804,-33.993,-100.023,166.251,52.186,159.437
C04412=1019.797,-34.242,-100.011,166.247,52.191,159.437
C04413=1019.792,-34.491,-99.999,166.245,52.196,159.438
C04414=1019.786,-34.741,-99.986,166.242,52.201,159.438
C04415=1019.781,-34.991,-99.975,166.239,52.206,159.438
C04416=1019.775,-35.241,-99.962,166.237,52.211,159.439
C04417=1019.770,-35.490,-99.950,166.234,52.216,159.439
C04418=1019.764,-35.740,-99.939,166.230,52.221,159.439
C04419=1019.758,-35.990,-99.927,166.228,52.226,159.440
C04420=1019.752,-36.239,-99.914,166.225,52.231,159.440
C04421=1019.747,-36.489,-99.902,166.221,52.236,159.440
C04422=1019.742,-36.738,-99.890,166.219,52.241,159.441
C04423=1019.735,-37.017,-99.877,166.216,52.246,159.441
C04424=1019.729,-37.294,-99.864,166.213,52.251,159.442
C04425=1019.723,-37.573,-99.851,166.209,52.258,159.442
C04426=1019.717,-37.850,-99.837,166.206,52.263,159.443
C04427=1019.711,-38.100,-99.825,166.204,52.267,159.443
C04428=1019.706,-38.350,-99.813,166.201,52.273,159.443
C04429=1019.700,-38.600,-99.801,166.198,52.278,159.444
C04430=1019.694,-38.849,-99.789,166.195,52.282,159.444
C04431=1019.688,-39.099,-99.777,166.192,52.287,159.444
C04432=1019.683,-39.349,-99.765,166.189,52.293,159.445
C04433=1019.677,-39.598,-99.754,166.186,52.297,159.445
C04434=1019.671,-39.848,-99.742,166.183,52.302,159.445
C04435=1019.666,-40.098,-99.730,166.180,52.308,159.446
C04436=1019.660,-40.347,-99.718,166.177,52.313,159.446
C04437=1019.655,-40.597,-99.707,166.175,52.318,159.447
C04438=1019.649,-40.847,-99.696,166.172,52.323,159.447
C04439=1019.643,-41.096,-99.683,166.168,52.328,159.447
C04440=1019.637,-41.346,-99.673,166.166,52.333,159.448
C04441=1019.631,-41.596,-99.660,166.163,52.338,159.448
C04442=1019.626,-41.845,-99.649,166.160,52.343,159.448
C04443=1019.621,-42.095,-99.638,166.157,52.348,159.449
C04444=1019.614,-42.345,-99.626,166.155,52.353,159.449
C04445=1019.609,-42.595,-99.614,166.152,52.359,159.449
C04446=1019.604,-42.844,-99.602,166.148,52.363,159.450
C04447=1019.597,-43.094,-99.591,166.146,52.368,159.450
C04448=1019.592,-43.344,-99.579,166.143,52.373,159.451
C04449=1019.586,-43.593,-99.568,166.139,52.378,159.451
C04450=1019.581,-43.843,-99.556,166.136,52.383,159.451
C04451=1019.575,-44.093,-99.545,166.134,52.388,159.452
C04452=1019.570,-44.342,-99.533,166.131,52.393,159.452
C04453=1019.564,-44.591,-99.522,166.128,52.398,159.452
C04454=1019.558,-44.842,-99.510,166.126,52.403,159.453
C04455=1019.552,-45.091,-99.499,166.122,52.408,159.453
C04456=1019.547,-45.340,-99.487,166.119,52.413,159.453
C04457=1019.541,-45.591,-99.476,166.117,52.418,159.454
C04458=1019.536,-45.840,-99.464,166.113,52.423,159.454
C04459=1019.531,-46.090,-99.452,166.110,52.428,159.454
C04460=1019.525,-46.339,-99.441,166.108,52.433,159.455
C04461=1019.519,-46.590,-99.429,166.105,52.438,159.455
C04462=1019.513,-46.838,-99.418,166.102,52.443,159.455
C04463=1019.508,-47.088,-99.406,166.100,52.448,159.456
C04464=1019.503,-47.338,-99.396,166.096,52.453,159.456
C04465=1019.497,-47.588,-99.384,166.093,52.458,159.456
C04466=1019.491,-47.838,-99.373,166.090,52.463,159.456
C04467=1019.486,-48.087,-99.361,166.088,52.468,159.457
C04468=1019.480,-48.336,-99.350,166.085,52.473,159.457
C04469=1019.475,-48.587,-99.338,166.081,52.478,159.457
C04470=1019.469,-48.836,-99.327,166.079,52.483,159.458
C04471=1019.464,-49.086,-99.316,166.075,52.487,159.458
C04472=1019.458,-49.335,-99.304,166.073,52.492,159.459
C04473=1019.453,-49.585,-99.292,166.070,52.497,159.459
C04474=1019.446,-49.835,-99.281,166.067,52.502,159.459
C04475=1019.441,-50.085,-99.270,166.064,52.507,159.459
C04476=1019.436,-50.334,-99.259,166.061,52.512,159.460
C04477=1019.431,-50.584,-99.247,166.058,52.517,159.460
C04478=1019.425,-50.833,-99.236,166.056,52.522,159.460
C04479=1019.420,-51.083,-99.224,166.053,52.527,159.461
C04480=1019.413,-51.333,-99.213,166.049,52.532,159.461
C04481=1019.408,-51.583,-99.203,166.046,52.537,159.461
C04482=1019.402,-51.833,-99.192,166.043,52.542,159.462
C04483=1019.396,-52.082,-99.181,166.041,52.547,159.462
C04484=1019.391,-52.332,-99.170,166.038,52.553,159.463
C04485=1019.385,-52.581,-99.159,166.034,52.557,159.463
C04486=1019.379,-52.832,-99.148,166.031,52.563,159.463
C04487=1019.373,-53.110,-99.136,166.029,52.569,159.464
C04488=1019.366,-53.387,-99.124,166.026,52.574,159.464
C04489=1019.360,-53.666,-99.111,166.021,52.580,159.464
C04490=1019.354,-53.944,-99.100,166.018,52.585,159.465
C04491=1019.348,-54.194,-99.089,166.015,52.591,159.465
C04492=1019.342,-54.443,-99.078,166.012,52.596,159.465
C04493=1019.337,-54.693,-99.066,166.010,52.601,159.466
C04494=1019.331,-54.943,-99.055,166.007,52.606,159.466
C04495=1019.325,-55.193,-99.045,166.004,52.611,159.466
///RCONF 1,0,0,1,0,0,0,0,0,0,0,0,0,0,0,0,0,0,0,0,0,0,0,0
C04496=1019.320,-55.443,-99.034,166.001,52.616,159.467
C04497=1019.314,-55.692,-99.023,165.997,52.621,159.467
C04498=1019.308,-55.942,-99.012,165.995,52.626,159.467
C04499=1019.302,-56.191,-99.001,165.992,52.631,159.468
C04500=1019.297,-56.442,-98.991,165.989,52.637,159.468
C04501=1019.291,-56.691,-98.980,165.985,52.641,159.468
C04502=1019.286,-56.941,-98.969,165.983,52.646,159.469
C04503=1019.281,-57.190,-98.958,165.980,52.652,159.469
C04504=1019.275,-57.440,-98.947,165.977,52.657,159.469
C04505=1019.269,-57.690,-98.937,165.974,52.662,159.470
C04506=1019.264,-57.939,-98.926,165.972,52.667,159.470
C04507=1019.258,-58.189,-98.915,165.968,52.672,159.470
C04508=1019.252,-58.438,-98.904,165.965,52.677,159.471
C04509=1019.247,-58.688,-98.894,165.962,52.682,159.471
C04510=1019.241,-58.938,-98.883,165.960,52.687,159.471
C04511=1019.235,-59.187,-98.872,165.957,52.692,159.472
C04512=1019.231,-59.438,-98.862,165.954,52.697,159.472
C04513=1019.225,-59.687,-98.851,165.950,52.702,159.472
C04514=1019.219,-59.937,-98.840,165.948,52.707,159.473
C04515=1019.213,-60.186,-98.829,165.945,52.712,159.473
C04516=1019.208,-60.436,-98.819,165.941,52.717,159.473
C04517=1019.202,-60.686,-98.808,165.938,52.722,159.474
C04518=1019.196,-60.935,-98.797,165.936,52.727,159.474
C04519=1019.191,-61.186,-98.787,165.933,52.732,159.474
C04520=1019.185,-61.435,-98.776,165.929,52.737,159.475
C04521=1019.180,-61.685,-98.766,165.926,52.742,159.475
C04522=1019.174,-61.935,-98.755,165.924,52.747,159.475
C04523=1019.168,-62.184,-98.744,165.921,52.752,159.476
C04524=1019.164,-62.435,-98.733,165.918,52.757,159.476
C04525=1019.158,-62.684,-98.723,165.914,52.762,159.476
C04526=1019.152,-62.934,-98.712,165.912,52.767,159.477
C04527=1019.147,-63.184,-98.701,165.909,52.772,159.477
C04528=1019.141,-63.433,-98.691,165.906,52.777,159.477
C04529=1019.136,-63.683,-98.680,165.903,52.782,159.477
C04530=1019.130,-63.933,-98.670,165.900,52.787,159.478
C04531=1019.125,-64.182,-98.660,165.897,52.792,159.478
C04532=1019.119,-64.432,-98.649,165.894,52.797,159.478
C04533=1019.113,-64.681,-98.638,165.892,52.802,159.479
C04534=1019.108,-64.931,-98.628,165.888,52.806,159.479
C04535=1019.102,-65.181,-98.617,165.885,52.812,159.479
C04536=1019.097,-65.431,-98.607,165.882,52.816,159.479
C04537=1019.091,-65.680,-98.596,165.880,52.822,159.480
C04538=1019.086,-65.931,-98.585,165.876,52.826,159.480
C04539=1019.081,-66.180,-98.575,165.873,52.832,159.480
C04540=1019.076,-66.430,-98.565,165.871,52.836,159.481
C04541=1019.070,-66.679,-98.554,165.868,52.841,159.481
C04542=1019.065,-66.929,-98.543,165.864,52.846,159.481
C04543=1019.059,-67.179,-98.533,165.861,52.851,159.482
C04544=1019.054,-67.429,-98.522,165.859,52.856,159.482
C04545=1019.049,-67.678,-98.513,165.856,52.861,159.482
C04546=1019.043,-67.928,-98.502,165.852,52.866,159.482
C04547=1019.038,-68.178,-98.492,165.850,52.871,159.483
C04548=1019.032,-68.427,-98.481,165.847,52.875,159.483
C04549=1019.026,-68.677,-98.471,165.843,52.880,159.483
C04550=1019.021,-68.926,-98.460,165.840,52.886,159.483
C04551=1019.016,-69.206,-98.449,165.837,52.891,159.484
C04552=1019.010,-69.486,-98.437,165.834,52.896,159.484
C04553=1019.003,-69.765,-98.425,165.831,52.902,159.485
C04554=1018.997,-70.045,-98.413,165.827,52.907,159.485
C04555=1018.992,-70.294,-98.404,165.824,52.912,159.485
C04556=1018.986,-70.544,-98.393,165.821,52.917,159.485
C04557=1018.981,-70.794,-98.382,165.818,52.922,159.485
C04558=1018.975,-71.044,-98.372,165.815,52.926,159.486
C04559=1018.970,-71.293,-98.362,165.812,52.932,159.486
C04560=1018.965,-71.543,-98.352,165.809,52.936,159.486
C04561=1018.959,-71.793,-98.341,165.807,52.941,159.487
C04562=1018.954,-72.043,-98.331,165.803,52.946,159.487
C04563=1018.950,-72.292,-98.320,165.800,52.951,159.487
C04564=1018.944,-72.542,-98.310,165.798,52.956,159.488
C04565=1018.938,-72.792,-98.299,165.794,52.960,159.488
C04566=1018.934,-73.041,-98.289,165.791,52.965,159.488
C04567=1018.928,-73.291,-98.279,165.789,52.970,159.488
C04568=1018.923,-73.541,-98.269,165.786,52.975,159.488
C04569=1018.918,-73.790,-98.259,165.782,52.980,159.489
C04570=1018.912,-74.040,-98.248,165.780,52.985,159.489
C04571=1018.907,-74.290,-98.238,165.777,52.989,159.489
C04572=1018.901,-74.541,-98.228,165.774,52.995,159.490
C04573=1018.896,-74.789,-98.218,165.770,52.999,159.490
C04574=1018.890,-75.039,-98.208,165.768,53.004,159.490
C04575=1018.884,-75.289,-98.198,165.765,53.009,159.490
C04576=1018.880,-75.539,-98.188,165.762,53.015,159.491
C04577=1018.873,-75.788,-98.178,165.758,53.019,159.491
C04578=1018.868,-76.039,-98.168,165.756,53.024,159.491
C04579=1018.863,-76.288,-98.158,165.753,53.030,159.492
C04580=1018.858,-76.538,-98.148,165.750,53.034,159.492
C04581=1018.852,-76.787,-98.139,165.747,53.040,159.492
C04582=1018.847,-77.037,-98.129,165.744,53.044,159.492
C04583=1018.841,-77.287,-98.119,165.741,53.050,159.493
C04584=1018.837,-77.537,-98.109,165.738,53.054,159.493
C04585=1018.830,-77.787,-98.099,165.735,53.060,159.493
C04586=1018.826,-78.036,-98.090,165.731,53.064,159.493
C04587=1018.820,-78.286,-98.079,165.729,53.069,159.494
C04588=1018.815,-78.536,-98.069,165.726,53.074,159.494
C04589=1018.809,-78.785,-98.060,165.723,53.080,159.494
C04590=1018.804,-79.035,-98.050,165.719,53.084,159.495
C04591=1018.799,-79.285,-98.040,165.717,53.089,159.495
C04592=1018.793,-79.535,-98.031,165.714,53.094,159.495
C04593=1018.787,-79.785,-98.020,165.711,53.099,159.496
C04594=1018.782,-80.034,-98.011,165.707,53.104,159.496
C04595=1018.777,-80.284,-98.000,165.705,53.108,159.496
C04596=1018.771,-80.533,-97.991,165.702,53.114,159.496
C04597=1018.766,-80.783,-97.981,165.699,53.119,159.497
C04598=1018.761,-81.033,-97.973,165.695,53.124,159.497
C04599=1018.755,-81.283,-97.962,165.692,53.129,159.497
C04600=1018.750,-81.532,-97.953,165.689,53.135,159.497
C04601=1018.743,-81.782,-97.944,165.687,53.139,159.498
C04602=1018.738,-82.033,-97.934,165.684,53.145,159.498
C04603=1018.733,-82.282,-97.925,165.681,53.150,159.498
C04604=1018.727,-82.532,-97.915,165.677,53.155,159.499
C04605=1018.722,-82.781,-97.906,165.674,53.160,159.499
C04606=1018.717,-83.032,-97.896,165.671,53.166,159.499
C04607=1018.711,-83.281,-97.887,165.668,53.170,159.499
C04608=1018.706,-83.531,-97.877,165.666,53.175,159.500
C04609=1018.700,-83.780,-97.868,165.662,53.180,159.500
C04610=1018.695,-84.031,-97.858,165.659,53.186,159.500
C04611=1018.689,-84.280,-97.849,165.656,53.191,159.501
C04612=1018.684,-84.529,-97.840,165.653,53.196,159.501
C04613=1018.679,-84.780,-97.830,165.650,53.201,159.501
C04614=1018.673,-85.029,-97.821,165.647,53.205,159.501
C04615=1018.667,-85.311,-97.810,165.644,53.212,159.502
C04616=1018.661,-85.592,-97.799,165.641,53.217,159.502
C04617=1018.654,-85.873,-97.789,165.637,53.223,159.502
C04618=1018.649,-86.156,-97.779,165.634,53.229,159.503
C04619=1018.643,-86.405,-97.769,165.631,53.234,159.503
C04620=1018.638,-86.655,-97.759,165.627,53.239,159.503
C04621=1018.633,-86.904,-97.751,165.624,53.244,159.504
C04622=1018.628,-87.154,-97.741,165.622,53.249,159.504
C04623=1018.622,-87.404,-97.731,165.619,53.254,159.504
C04624=1018.617,-87.654,-97.722,165.615,53.259,159.504
C04625=1018.611,-87.904,-97.713,165.612,53.264,159.505
C04626=1018.606,-88.153,-97.704,165.609,53.269,159.505
C04627=1018.601,-88.403,-97.695,165.607,53.274,159.505
C04628=1018.595,-88.653,-97.686,165.603,53.279,159.505
C04629=1018.590,-88.902,-97.676,165.600,53.284,159.506
C04630=1018.584,-89.152,-97.666,165.597,53.289,159.506
C04631=1018.579,-89.402,-97.657,165.594,53.294,159.506
C04632=1018.574,-89.651,-97.648,165.591,53.299,159.507
C04633=1018.568,-89.902,-97.639,165.588,53.304,159.507
C04634=1018.563,-90.151,-97.629,165.585,53.309,159.507
C04635=1018.558,-90.401,-97.621,165.582,53.314,159.507
C04636=1018.552,-90.651,-97.611,165.578,53.319,159.507
C04637=1018.547,-90.901,-97.602,165.576,53.324,159.508
C04638=1018.542,-91.150,-97.592,165.573,53.329,159.508
C04639=1018.536,-91.401,-97.584,165.570,53.334,159.508
C04640=1018.531,-91.650,-97.574,165.566,53.339,159.509
C04641=1018.526,-91.900,-97.565,165.563,53.344,159.509
C04642=1018.521,-92.149,-97.557,165.561,53.349,159.509
C04643=1018.516,-92.400,-97.547,165.558,53.354,159.510
C04644=1018.510,-92.649,-97.538,165.555,53.359,159.510
C04645=1018.505,-92.898,-97.529,165.552,53.364,159.510
C04646=1018.500,-93.149,-97.520,165.549,53.369,159.510
C04647=1018.494,-93.398,-97.510,165.546,53.374,159.511
C04648=1018.490,-93.648,-97.501,165.543,53.379,159.511
C04649=1018.484,-93.898,-97.493,165.539,53.384,159.511
C04650=1018.479,-94.148,-97.483,165.537,53.389,159.511
C04651=1018.474,-94.398,-97.474,165.534,53.394,159.511
C04652=1018.468,-94.647,-97.465,165.531,53.399,159.512
C04653=1018.463,-94.897,-97.456,165.527,53.404,159.512
C04654=1018.458,-95.147,-97.447,165.525,53.408,159.512
C04655=1018.453,-95.397,-97.437,165.522,53.414,159.513
C04656=1018.448,-95.646,-97.429,165.519,53.418,159.513
C04657=1018.442,-95.896,-97.420,165.516,53.424,159.513
C04658=1018.437,-96.146,-97.410,165.513,53.428,159.513
C04659=1018.432,-96.396,-97.402,165.510,53.433,159.513
C04660=1018.427,-96.646,-97.393,165.507,53.438,159.514
C04661=1018.421,-96.895,-97.383,165.503,53.443,159.514
C04662=1018.416,-97.145,-97.375,165.501,53.448,159.514
C04663=1018.412,-97.395,-97.366,165.498,53.453,159.514
C04664=1018.406,-97.645,-97.357,165.494,53.458,159.515
C04665=1018.401,-97.895,-97.347,165.491,53.463,159.515
C04666=1018.396,-98.144,-97.339,165.488,53.468,159.515
C04667=1018.390,-98.394,-97.330,165.486,53.473,159.515
C04668=1018.385,-98.644,-97.322,165.482,53.478,159.516
C04669=1018.380,-98.893,-97.313,165.479,53.483,159.516
C04670=1018.374,-99.144,-97.304,165.476,53.488,159.516
C04671=1018.369,-99.394,-97.296,165.473,53.493,159.516
C04672=1018.363,-99.643,-97.287,165.470,53.499,159.517
C04673=1018.359,-99.893,-97.278,165.468,53.503,159.517
C04674=1018.353,-100.142,-97.269,165.465,53.509,159.517
C04675=1018.348,-100.392,-97.261,165.461,53.513,159.517
C04676=1018.343,-100.642,-97.252,165.458,53.519,159.518
C04677=1018.338,-100.892,-97.244,165.455,53.524,159.518
C04678=1018.332,-101.142,-97.235,165.452,53.529,159.518
C04679=1018.327,-101.398,-97.226,165.449,53.534,159.518
C04680=1018.322,-101.654,-97.217,165.446,53.539,159.519
C04681=1018.316,-101.911,-97.209,165.443,53.545,159.519
C04682=1018.311,-102.167,-97.200,165.440,53.549,159.519
C04683=1018.306,-102.417,-97.191,165.437,53.555,159.520
C04684=1018.300,-102.667,-97.183,165.433,53.559,159.520
C04685=1018.295,-102.916,-97.174,165.430,53.565,159.520
C04686=1018.291,-103.166,-97.165,165.427,53.570,159.520
C04687=1018.285,-103.417,-97.157,165.425,53.575,159.521
C04688=1018.279,-103.667,-97.148,165.422,53.580,159.521
C04689=1018.274,-103.916,-97.140,165.419,53.585,159.521
C04690=1018.269,-104.166,-97.131,165.415,53.590,159.521
C04691=1018.264,-104.416,-97.123,165.412,53.595,159.522
C04692=1018.258,-104.665,-97.114,165.410,53.600,159.522
C04693=1018.253,-104.915,-97.106,165.406,53.604,159.522
C04694=1018.248,-105.165,-97.097,165.403,53.610,159.522
C04695=1018.242,-105.442,-97.087,165.400,53.615,159.523
C04696=1018.237,-105.719,-97.078,165.396,53.621,159.523
C04697=1018.231,-105.996,-97.069,165.393,53.627,159.523
C04698=1018.225,-106.273,-97.060,165.390,53.632,159.523
C04699=1018.219,-106.522,-97.051,165.387,53.637,159.524
C04700=1018.215,-106.773,-97.043,165.384,53.642,159.524
C04701=1018.209,-107.022,-97.035,165.380,53.647,159.524
C04702=1018.204,-107.272,-97.026,165.379,53.652,159.524
C04703=1018.199,-107.522,-97.017,165.375,53.657,159.525
C04704=1018.194,-107.772,-97.009,165.372,53.663,159.525
C04705=1018.189,-108.022,-97.001,165.369,53.667,159.525
C04706=1018.183,-108.271,-96.993,165.366,53.673,159.525
C04707=1018.179,-108.520,-96.985,165.362,53.678,159.525
C04708=1018.173,-108.770,-96.977,165.360,53.683,159.526
C04709=1018.168,-109.021,-96.969,165.357,53.688,159.526
C04710=1018.163,-109.270,-96.960,165.354,53.693,159.526
C04711=1018.158,-109.520,-96.952,165.350,53.698,159.526
C04712=1018.153,-109.770,-96.943,165.347,53.703,159.527
C04713=1018.148,-110.020,-96.936,165.344,53.708,159.527
C04714=1018.142,-110.270,-96.927,165.342,53.713,159.527
C04715=1018.136,-110.519,-96.919,165.339,53.718,159.528
C04716=1018.131,-110.769,-96.911,165.336,53.723,159.528
C04717=1018.126,-111.019,-96.903,165.332,53.728,159.528
C04718=1018.121,-111.268,-96.895,165.329,53.734,159.528
C04719=1018.116,-111.519,-96.887,165.326,53.738,159.528
C04720=1018.111,-111.768,-96.879,165.324,53.744,159.529
C04721=1018.106,-112.019,-96.871,165.320,53.748,159.529
C04722=1018.101,-112.268,-96.862,165.317,53.754,159.529
C04723=1018.096,-112.518,-96.854,165.314,53.759,159.529
C04724=1018.090,-112.768,-96.847,165.311,53.764,159.530
C04725=1018.085,-113.017,-96.838,165.309,53.769,159.530
C04726=1018.080,-113.267,-96.831,165.306,53.774,159.530
C04727=1018.075,-113.517,-96.822,165.302,53.779,159.530
C04728=1018.070,-113.767,-96.814,165.299,53.784,159.531
C04729=1018.065,-114.017,-96.806,165.296,53.789,159.531
C04730=1018.060,-114.266,-96.798,165.294,53.794,159.531
C04731=1018.055,-114.517,-96.790,165.291,53.799,159.531
C04732=1018.049,-114.766,-96.782,165.287,53.804,159.532
C04733=1018.044,-115.016,-96.774,165.284,53.809,159.532
C04734=1018.039,-115.266,-96.766,165.281,53.815,159.532
C04735=1018.035,-115.516,-96.759,165.279,53.819,159.532
C04736=1018.029,-115.765,-96.750,165.276,53.825,159.533
C04737=1018.024,-116.015,-96.743,165.272,53.829,159.533
C04738=1018.018,-116.265,-96.734,165.269,53.835,159.533
C04739=1018.014,-116.515,-96.727,165.266,53.840,159.533
C04740=1018.009,-116.765,-96.719,165.263,53.845,159.534
C04741=1018.003,-117.014,-96.711,165.261,53.850,159.534
C04742=1017.998,-117.265,-96.704,165.258,53.855,159.534
C04743=1017.993,-117.548,-96.694,165.254,53.861,159.534
C04744=1017.986,-117.831,-96.685,165.251,53.867,159.535
C04745=1017.981,-118.115,-96.677,165.247,53.872,159.535
C04746=1017.975,-118.399,-96.668,165.244,53.878,159.535
C04747=1017.970,-118.649,-96.660,165.240,53.883,159.535
C04748=1017.965,-118.898,-96.653,165.237,53.888,159.536
C04749=1017.960,-119.148,-96.645,165.235,53.893,159.536
C04750=1017.955,-119.398,-96.637,165.232,53.898,159.536
C04751=1017.950,-119.647,-96.629,165.228,53.903,159.536
C04752=1017.944,-119.897,-96.622,165.226,53.909,159.537
C04753=1017.939,-120.148,-96.614,165.222,53.913,159.537
C04754=1017.935,-120.397,-96.606,165.219,53.919,159.537
C04755=1017.929,-120.647,-96.599,165.217,53.923,159.537
C04756=1017.924,-120.897,-96.591,165.214,53.929,159.538
C04757=1017.920,-121.147,-96.584,165.210,53.934,159.538
C04758=1017.914,-121.396,-96.576,165.207,53.939,159.538
C04759=1017.909,-121.647,-96.568,165.204,53.944,159.538
C04760=1017.904,-121.896,-96.561,165.202,53.949,159.539
C04761=1017.899,-122.146,-96.553,165.199,53.954,159.539
C04762=1017.893,-122.396,-96.545,165.196,53.959,159.539
C04763=1017.889,-122.646,-96.538,165.192,53.964,159.539
C04764=1017.883,-122.896,-96.530,165.190,53.969,159.540
C04765=1017.879,-123.145,-96.523,165.187,53.974,159.540
C04766=1017.874,-123.396,-96.515,165.184,53.980,159.540
C04767=1017.868,-123.645,-96.507,165.181,53.984,159.540
C04768=1017.864,-123.895,-96.500,165.177,53.989,159.540
C04769=1017.859,-124.145,-96.492,165.175,53.994,159.541
C04770=1017.854,-124.394,-96.485,165.172,53.999,159.541
C04771=1017.849,-124.645,-96.478,165.169,54.005,159.541
C04772=1017.843,-124.895,-96.470,165.165,54.009,159.541
C04773=1017.839,-125.144,-96.463,165.162,54.015,159.542
C04774=1017.833,-125.394,-96.456,165.160,54.019,159.542
C04775=1017.829,-125.644,-96.448,165.157,54.025,159.542
C04776=1017.823,-125.893,-96.441,165.154,54.030,159.542
C04777=1017.818,-126.143,-96.433,165.151,54.035,159.542
C04778=1017.813,-126.393,-96.426,165.147,54.040,159.543
C04779=1017.808,-126.643,-96.419,165.144,54.046,159.543
C04780=1017.803,-126.893,-96.411,165.142,54.050,159.543
C04781=1017.798,-127.142,-96.404,165.139,54.056,159.543
C04782=1017.792,-127.392,-96.397,165.136,54.060,159.544
C04783=1017.788,-127.642,-96.389,165.133,54.066,159.544
C04784=1017.782,-127.892,-96.382,165.129,54.071,159.544
C04785=1017.778,-128.142,-96.375,165.127,54.076,159.544
C04786=1017.774,-128.391,-96.367,165.124,54.081,159.545
C04787=1017.770,-128.640,-96.359,165.121,54.084,159.545
C04788=1017.765,-128.891,-96.350,165.118,54.088,159.545
C04789=1017.762,-129.140,-96.340,165.116,54.091,159.545
C04790=1017.759,-129.389,-96.330,165.113,54.093,159.544
C04791=1017.757,-129.639,-96.319,165.111,54.094,159.544
C04792=1017.755,-129.888,-96.308,165.108,54.096,159.544
C04793=1017.752,-130.138,-96.295,165.106,54.097,159.543
C04794=1017.751,-130.388,-96.283,165.103,54.097,159.543
C04795=1017.751,-130.638,-96.269,165.101,54.097,159.542
C04796=1017.750,-130.887,-96.256,165.099,54.096,159.542
C04797=1017.750,-131.138,-96.241,165.096,54.094,159.541
C04798=1017.751,-131.387,-96.226,165.094,54.092,159.540
C04799=1017.751,-131.637,-96.211,165.092,54.090,159.539
C04800=1017.753,-131.887,-96.194,165.090,54.086,159.538
C04801=1017.754,-132.137,-96.178,165.088,54.083,159.537
C04802=1017.756,-132.385,-96.161,165.086,54.079,159.536
C04803=1017.759,-132.635,-96.143,165.085,54.074,159.535
C04804=1017.762,-132.886,-96.125,165.083,54.069,159.533
C04805=1017.765,-133.135,-96.106,165.082,54.063,159.532
C04806=1017.769,-133.384,-96.085,165.080,54.056,159.531
C04807=1017.507,-133.410,-96.466,165.038,54.403,159.582
C04808=1017.503,-133.162,-96.486,165.040,54.409,159.583
C04809=1017.500,-132.912,-96.505,165.042,54.415,159.585
C04810=1017.497,-132.662,-96.524,165.043,54.420,159.586
C04811=1017.495,-132.412,-96.542,165.045,54.425,159.587
C04812=1017.493,-132.162,-96.559,165.047,54.429,159.588
C04813=1017.491,-131.913,-96.576,165.049,54.433,159.589
C04814=1017.490,-131.663,-96.591,165.050,54.436,159.590
C04815=1017.489,-131.413,-96.607,165.053,54.439,159.591
C04816=1017.488,-131.164,-96.622,165.055,54.441,159.592
C04817=1017.489,-130.914,-96.636,165.057,54.442,159.593
C04818=1017.489,-130.664,-96.650,165.060,54.443,159.594
C04819=1017.490,-130.414,-96.664,165.062,54.443,159.594
C04820=1017.491,-130.164,-96.677,165.064,54.443,159.594
C04821=1017.493,-129.915,-96.688,165.066,54.442,159.595
C04822=1017.495,-129.665,-96.700,165.069,54.441,159.595
C04823=1017.497,-129.416,-96.710,165.072,54.439,159.596
C04824=1017.500,-129.166,-96.721,165.074,54.437,159.596
C04825=1017.504,-128.916,-96.731,165.078,54.434,159.596
C04826=1017.508,-128.667,-96.739,165.079,54.430,159.596
C04827=1017.512,-128.417,-96.748,165.083,54.426,159.596
C04828=1017.516,-128.168,-96.756,165.086,54.422,159.596
C04829=1017.521,-127.919,-96.764,165.089,54.416,159.595
C04830=1017.526,-127.669,-96.771,165.092,54.411,159.595
C04831=1017.531,-127.419,-96.778,165.095,54.406,159.595
C04832=1017.536,-127.170,-96.785,165.097,54.401,159.595
C04833=1017.541,-126.919,-96.793,165.100,54.396,159.594
C04834=1017.546,-126.670,-96.800,165.103,54.390,159.594
C04835=1017.551,-126.420,-96.807,165.106,54.385,159.594
C04836=1017.556,-126.170,-96.814,165.109,54.380,159.594
C04837=1017.561,-125.920,-96.822,165.113,54.375,159.593
C04838=1017.566,-125.671,-96.829,165.116,54.369,159.593
C04839=1017.571,-125.420,-96.837,165.118,54.364,159.593
C04840=1017.577,-125.170,-96.844,165.122,54.359,159.593
C04841=1017.581,-124.921,-96.851,165.124,54.354,159.592
C04842=1017.587,-124.671,-96.858,165.127,54.348,159.592
C04843=1017.591,-124.421,-96.866,165.130,54.343,159.592
C04844=1017.596,-124.171,-96.873,165.133,54.338,159.592
C04845=1017.601,-123.921,-96.880,165.136,54.333,159.591
C04846=1017.606,-123.671,-96.888,165.139,54.327,159.591
C04847=1017.611,-123.422,-96.895,165.143,54.323,159.591
C04848=1017.616,-123.172,-96.903,165.145,54.317,159.591
C04849=1017.621,-122.922,-96.911,165.148,54.313,159.590
C04850=1017.626,-122.672,-96.918,165.151,54.307,159.590
C04851=1017.631,-122.422,-96.926,165.154,54.302,159.590
C04852=1017.636,-122.172,-96.933,165.157,54.297,159.590
C04853=1017.641,-121.922,-96.940,165.160,54.291,159.589
C04854=1017.647,-121.673,-96.949,165.163,54.286,159.589
C04855=1017.651,-121.423,-96.956,165.165,54.281,159.589
C04856=1017.657,-121.173,-96.963,165.169,54.276,159.589
C04857=1017.661,-120.923,-96.971,165.172,54.271,159.588
C04858=1017.666,-120.674,-96.979,165.175,54.266,159.588
C04859=1017.672,-120.424,-96.986,165.178,54.260,159.588
C04860=1017.676,-120.174,-96.994,165.181,54.255,159.588
C04861=1017.681,-119.924,-97.002,165.184,54.250,159.588
C04862=1017.687,-119.674,-97.010,165.187,54.244,159.587
C04863=1017.692,-119.425,-97.017,165.190,54.240,159.587
C04864=1017.697,-119.174,-97.025,165.192,54.234,159.587
C04865=1017.702,-118.924,-97.032,165.196,54.230,159.586
C04866=1017.707,-118.675,-97.040,165.199,54.224,159.586
C04867=1017.712,-118.425,-97.048,165.202,54.218,159.586
C04868=1017.718,-118.142,-97.056,165.206,54.213,159.586
C04869=1017.723,-117.858,-97.065,165.209,54.207,159.585
C04870=1017.730,-117.575,-97.074,165.213,54.201,159.585
C04871=1017.735,-117.291,-97.083,165.215,54.195,159.585
C04872=1017.740,-117.041,-97.091,165.218,54.190,159.585
C04873=1017.746,-116.792,-97.098,165.221,54.184,159.584
C04874=1017.751,-116.542,-97.106,165.225,54.180,159.584
C04875=1017.755,-116.291,-97.114,165.228,54.174,159.584
C04876=1017.760,-116.042,-97.122,165.231,54.169,159.584
C04877=1017.766,-115.792,-97.129,165.234,54.164,159.583
C04878=1017.771,-115.542,-97.138,165.236,54.159,159.583
C04879=1017.776,-115.292,-97.146,165.239,54.154,159.583
C04880=1017.781,-115.043,-97.154,165.242,54.148,159.582
C04881=1017.786,-114.793,-97.161,165.245,54.143,159.582
C04882=1017.791,-114.543,-97.169,165.249,54.138,159.582
C04883=1017.797,-114.293,-97.177,165.252,54.132,159.582
C04884=1017.801,-114.044,-97.185,165.255,54.128,159.582
C04885=1017.806,-113.794,-97.193,165.258,54.122,159.581
C04886=1017.812,-113.544,-97.201,165.260,54.118,159.581
C04887=1017.816,-113.294,-97.209,165.263,54.112,159.581
C04888=1017.822,-113.044,-97.218,165.267,54.107,159.581
C04889=1017.827,-112.795,-97.225,165.270,54.102,159.580
C04890=1017.832,-112.545,-97.233,165.272,54.096,159.580
C04891=1017.837,-112.295,-97.241,165.276,54.091,159.580
C04892=1017.842,-112.045,-97.249,165.279,54.086,159.579
C04893=1017.848,-111.795,-97.258,165.282,54.081,159.579
C04894=1017.852,-111.545,-97.265,165.285,54.075,159.579
C04895=1017.857,-111.296,-97.274,165.287,54.070,159.579
C04896=1017.862,-111.045,-97.281,165.290,54.066,159.578
C04897=1017.868,-110.796,-97.289,165.293,54.060,159.578
C04898=1017.873,-110.546,-97.298,165.297,54.055,159.578
C04899=1017.878,-110.296,-97.306,165.300,54.050,159.578
C04900=1017.884,-110.046,-97.314,165.303,54.044,159.577
C04901=1017.888,-109.797,-97.322,165.306,54.039,159.577
C04902=1017.893,-109.547,-97.330,165.309,54.034,159.577
C04903=1017.899,-109.297,-97.338,165.312,54.028,159.577
C04904=1017.904,-109.047,-97.347,165.315,54.023,159.576
C04905=1017.909,-108.797,-97.355,165.317,54.018,159.576
C04906=1017.914,-108.547,-97.363,165.321,54.014,159.576
C04907=1017.920,-108.298,-97.371,165.324,54.008,159.576
C04908=1017.925,-108.048,-97.379,165.327,54.002,159.575
C04909=1017.930,-107.798,-97.387,165.330,53.998,159.575
C04910=1017.936,-107.548,-97.396,165.333,53.992,159.575
C04911=1017.941,-107.299,-97.404,165.336,53.987,159.574
C04912=1017.945,-107.049,-97.412,165.339,53.982,159.574
C04913=1017.950,-106.799,-97.420,165.342,53.976,159.574
C04914=1017.956,-106.549,-97.429,165.346,53.972,159.574
C04915=1017.961,-106.300,-97.437,165.348,53.966,159.573
C04916=1017.965,-106.050,-97.446,165.351,53.962,159.573
C04917=1017.971,-105.800,-97.455,165.354,53.956,159.573
C04918=1017.976,-105.550,-97.462,165.357,53.951,159.573
C04919=1017.981,-105.300,-97.471,165.360,53.946,159.572
C04920=1017.986,-105.050,-97.479,165.363,53.940,159.572
C04921=1017.991,-104.801,-97.488,165.367,53.935,159.572
C04922=1017.997,-104.551,-97.496,165.370,53.930,159.572
C04923=1018.002,-104.301,-97.505,165.372,53.926,159.571
C04924=1018.007,-104.051,-97.513,165.375,53.920,159.571
C04925=1018.013,-103.802,-97.522,165.378,53.915,159.571
C04926=1018.018,-103.552,-97.530,165.381,53.910,159.571
C04927=1018.023,-103.302,-97.539,165.384,53.904,159.570
C04928=1018.027,-103.052,-97.547,165.388,53.899,159.570
C04929=1018.033,-102.802,-97.556,165.391,53.894,159.570
C04930=1018.038,-102.552,-97.564,165.393,53.888,159.570
C04931=1018.043,-102.302,-97.573,165.396,53.884,159.569
C04932=1018.049,-102.019,-97.583,165.400,53.878,159.569
C04933=1018.055,-101.735,-97.592,165.403,53.872,159.569
C04934=1018.061,-101.452,-97.602,165.406,53.866,159.568
C04935=1018.068,-101.169,-97.612,165.410,53.860,159.568
C04936=1018.072,-100.919,-97.621,165.413,53.855,159.568
C04937=1018.077,-100.669,-97.629,165.417,53.850,159.568
C04938=1018.083,-100.419,-97.638,165.419,53.845,159.567
C04939=1018.088,-100.169,-97.646,165.422,53.839,159.567
C04940=1018.093,-99.920,-97.655,165.425,53.834,159.567
C04941=1018.099,-99.670,-97.663,165.428,53.829,159.566
C04942=1018.104,-99.420,-97.672,165.431,53.823,159.566
C04943=1018.109,-99.171,-97.680,165.434,53.819,159.566
C04944=1018.115,-98.922,-97.689,165.437,53.813,159.566
C04945=1018.120,-98.671,-97.699,165.440,53.808,159.565
C04946=1018.125,-98.421,-97.707,165.444,53.803,159.565
C04947=1018.130,-98.171,-97.716,165.447,53.797,159.565
C04948=1018.136,-97.922,-97.724,165.450,53.792,159.564
C04949=1018.141,-97.672,-97.733,165.452,53.787,159.564
C04950=1018.145,-97.422,-97.742,165.455,53.782,159.564
C04951=1018.151,-97.172,-97.751,165.458,53.777,159.564
C04952=1018.156,-96.922,-97.760,165.461,53.772,159.563
C04953=1018.161,-96.672,-97.769,165.465,53.767,159.563
C04954=1018.167,-96.423,-97.777,165.468,53.761,159.563
C04955=1018.171,-96.173,-97.787,165.470,53.757,159.563
C04956=1018.177,-95.924,-97.796,165.473,53.752,159.562
C04957=1018.182,-95.673,-97.805,165.476,53.747,159.562
C04958=1018.187,-95.424,-97.814,165.479,53.741,159.562
C04959=1018.193,-95.174,-97.823,165.483,53.737,159.562
C04960=1018.197,-94.924,-97.832,165.485,53.731,159.561
C04961=1018.203,-94.675,-97.841,165.488,53.727,159.561
C04962=1018.207,-94.425,-97.850,165.491,53.721,159.561
C04963=1018.213,-94.174,-97.859,165.495,53.716,159.561
C04964=1018.219,-93.925,-97.868,165.498,53.711,159.560
C04965=1018.223,-93.675,-97.877,165.501,53.706,159.560
C04966=1018.228,-93.426,-97.886,165.504,53.701,159.560
C04967=1018.234,-93.175,-97.896,165.506,53.696,159.560
C04968=1018.243,-92.766,-97.910,165.511,53.687,159.559
C04969=1018.251,-92.356,-97.925,165.516,53.679,159.559
C04970=1018.260,-91.947,-97.940,165.521,53.671,159.558
C04971=1018.268,-91.537,-97.955,165.526,53.663,159.558
C04972=1018.274,-91.288,-97.964,165.529,53.657,159.557
C04973=1018.279,-91.038,-97.974,165.533,53.652,159.557
C04974=1018.284,-90.789,-97.983,165.536,53.647,159.557
C04975=1018.289,-90.539,-97.992,165.539,53.641,159.557
C04976=1018.294,-90.289,-98.000,165.542,53.637,159.557
C04977=1018.300,-90.039,-98.011,165.544,53.631,159.556
C04978=1018.305,-89.789,-98.019,165.547,53.627,159.556
C04979=1018.310,-89.540,-98.028,165.550,53.621,159.556
C04980=1018.316,-89.289,-98.038,165.553,53.616,159.555
C04981=1018.321,-89.040,-98.047,165.557,53.611,159.555
C04982=1018.326,-88.790,-98.056,165.560,53.606,159.555
C04983=1018.332,-88.540,-98.066,165.563,53.600,159.554
C04984=1018.336,-88.290,-98.075,165.566,53.595,159.554
C04985=1018.342,-88.041,-98.084,165.568,53.590,159.554
C04986=1018.348,-87.791,-98.093,165.571,53.585,159.553
C04987=1018.353,-87.541,-98.102,165.575,53.580,159.553
C04988=1018.359,-87.292,-98.112,165.577,53.575,159.553
C04989=1018.363,-87.041,-98.121,165.580,53.569,159.553
C04990=1018.369,-86.792,-98.130,165.584,53.564,159.553
C04991=1018.374,-86.542,-98.140,165.587,53.559,159.552
C04992=1018.383,-86.171,-98.154,165.591,53.551,159.552
C04993=1018.390,-85.799,-98.167,165.595,53.543,159.551
C04994=1018.398,-85.428,-98.181,165.600,53.535,159.551
C04995=1018.406,-85.057,-98.195,165.605,53.528,159.550
C04996=1018.412,-84.807,-98.205,165.608,53.523,159.550
C04997=1018.417,-84.557,-98.214,165.611,53.518,159.550
C04998=1018.423,-84.308,-98.223,165.614,53.512,159.550
C04999=1018.428,-84.058,-98.233,165.617,53.507,159.549
C05000=1018.434,-83.808,-98.242,165.620,53.502,159.549
C05001=1018.438,-83.558,-98.252,165.623,53.496,159.549
C05002=1018.445,-83.309,-98.261,165.625,53.491,159.548
C05003=1018.449,-83.059,-98.270,165.628,53.486,159.548
C05004=1018.455,-82.809,-98.280,165.632,53.481,159.548
C05005=1018.461,-82.560,-98.289,165.635,53.476,159.547
C05006=1018.465,-82.310,-98.298,165.638,53.470,159.547
C05007=1018.472,-82.060,-98.308,165.641,53.465,159.547
C05008=1018.476,-81.810,-98.318,165.644,53.460,159.547
C05009=1018.483,-81.561,-98.327,165.647,53.455,159.546
C05010=1018.487,-81.311,-98.336,165.650,53.449,159.546
C05011=1018.493,-81.061,-98.346,165.653,53.444,159.545
C05012=1018.498,-80.811,-98.356,165.657,53.439,159.545
C05013=1018.504,-80.562,-98.365,165.660,53.433,159.545
C05014=1018.509,-80.311,-98.375,165.663,53.428,159.545
C05015=1018.515,-80.062,-98.384,165.666,53.423,159.544
C05016=1018.520,-79.812,-98.394,165.668,53.418,159.544
C05017=1018.525,-79.562,-98.404,165.671,53.413,159.544
C05018=1018.531,-79.312,-98.413,165.674,53.408,159.544
C05019=1018.536,-79.063,-98.423,165.677,53.403,159.543
C05020=1018.542,-78.813,-98.433,165.680,53.397,159.543
C05021=1018.546,-78.564,-98.443,165.684,53.392,159.543
C05022=1018.553,-78.314,-98.453,165.686,53.387,159.542
C05023=1018.558,-78.064,-98.463,165.689,53.383,159.542
C05024=1018.563,-77.814,-98.473,165.692,53.377,159.542
C05025=1018.569,-77.564,-98.482,165.695,53.372,159.541
C05026=1018.574,-77.315,-98.492,165.699,53.367,159.541
C05027=1018.579,-77.065,-98.502,165.702,53.361,159.541
C05028=1018.584,-76.815,-98.512,165.704,53.356,159.540
C05029=1018.590,-76.566,-98.522,165.707,53.352,159.540
C05030=1018.596,-76.316,-98.532,165.710,53.346,159.540
C05031=1018.601,-76.066,-98.542,165.713,53.341,159.540
C05032=1018.606,-75.816,-98.552,165.717,53.336,159.539
C05033=1018.612,-75.566,-98.561,165.719,53.331,159.539
C05034=1018.617,-75.317,-98.571,165.722,53.325,159.539
C05035=1018.622,-75.067,-98.581,165.726,53.320,159.539
C05036=1018.627,-74.817,-98.591,165.728,53.315,159.538
C05037=1018.633,-74.568,-98.601,165.731,53.310,159.538
C05038=1018.639,-74.317,-98.611,165.734,53.305,159.538
C05039=1018.644,-74.068,-98.621,165.737,53.300,159.537
C05040=1018.649,-73.819,-98.631,165.741,53.295,159.537
C05041=1018.655,-73.568,-98.642,165.743,53.290,159.537
C05042=1018.660,-73.319,-98.651,165.746,53.285,159.536
C05043=1018.665,-73.069,-98.662,165.749,53.280,159.536
C05044=1018.671,-72.819,-98.672,165.753,53.275,159.536
C05045=1018.675,-72.570,-98.683,165.755,53.270,159.535
C05046=1018.680,-72.320,-98.693,165.758,53.265,159.535
C05047=1018.686,-72.069,-98.703,165.761,53.260,159.535
C05048=1018.691,-71.821,-98.714,165.765,53.255,159.535
C05049=1018.696,-71.571,-98.724,165.766,53.250,159.534
C05050=1018.702,-71.320,-98.734,165.770,53.245,159.534
C05051=1018.708,-71.071,-98.745,165.773,53.240,159.534
C05052=1018.712,-70.822,-98.755,165.776,53.235,159.534
C05053=1018.718,-70.571,-98.765,165.778,53.230,159.533
C05054=1018.723,-70.321,-98.775,165.782,53.225,159.533
C05055=1018.728,-70.073,-98.785,165.785,53.220,159.533
C05056=1018.734,-69.793,-98.797,165.788,53.215,159.532
C05057=1018.741,-69.513,-98.808,165.792,53.209,159.532
C05058=1018.746,-69.234,-98.820,165.795,53.203,159.532
C05059=1018.752,-68.955,-98.832,165.798,53.198,159.531
C05060=1018.758,-68.705,-98.843,165.801,53.192,159.531
C05061=1018.763,-68.455,-98.853,165.804,53.188,159.531
C05062=1018.768,-68.206,-98.863,165.807,53.182,159.530
C05063=1018.774,-67.956,-98.874,165.810,53.178,159.530
C05064=1018.779,-67.706,-98.884,165.813,53.173,159.530
C05065=1018.785,-67.456,-98.895,165.816,53.167,159.529
C05066=1018.791,-67.206,-98.905,165.819,53.162,159.529
C05067=1018.795,-66.957,-98.915,165.822,53.157,159.529
C05068=1018.801,-66.707,-98.925,165.825,53.153,159.529
C05069=1018.807,-66.457,-98.936,165.828,53.147,159.528
C05070=1018.812,-66.208,-98.946,165.831,53.142,159.528
C05071=1018.818,-65.958,-98.957,165.834,53.137,159.528
C05072=1018.823,-65.709,-98.967,165.837,53.132,159.527
C05073=1018.828,-65.459,-98.977,165.839,53.127,159.527
C05074=1018.834,-65.209,-98.988,165.843,53.122,159.527
C05075=1018.839,-64.959,-98.999,165.846,53.116,159.526
C05076=1018.845,-64.709,-99.010,165.849,53.112,159.526
C05077=1018.850,-64.459,-99.020,165.852,53.106,159.526
C05078=1018.856,-64.210,-99.031,165.854,53.101,159.525
C05079=1018.861,-63.960,-99.041,165.858,53.097,159.525
C05080=1018.866,-63.711,-99.052,165.861,53.091,159.525
C05081=1018.872,-63.461,-99.062,165.864,53.086,159.525
C05082=1018.877,-63.211,-99.073,165.867,53.081,159.524
C05083=1018.883,-62.961,-99.083,165.869,53.076,159.524
C05084=1018.889,-62.712,-99.094,165.872,53.071,159.524
C05085=1018.894,-62.462,-99.104,165.875,53.065,159.523
C05086=1018.900,-62.212,-99.115,165.879,53.061,159.523
C05087=1018.906,-61.963,-99.126,165.882,53.055,159.523
C05088=1018.910,-61.713,-99.135,165.885,53.050,159.522
C05089=1018.915,-61.463,-99.147,165.887,53.045,159.522
C05090=1018.921,-61.214,-99.158,165.890,53.040,159.522
C05091=1018.927,-60.964,-99.168,165.893,53.035,159.521
C05092=1018.932,-60.714,-99.179,165.896,53.029,159.521
C05093=1018.938,-60.464,-99.189,165.900,53.024,159.521
C05094=1018.943,-60.215,-99.200,165.903,53.019,159.520
C05095=1018.949,-59.965,-99.211,165.905,53.014,159.520
C05096=1018.955,-59.715,-99.221,165.908,53.009,159.520
C05097=1018.960,-59.466,-99.232,165.911,53.004,159.519
C05098=1018.966,-59.216,-99.243,165.914,52.998,159.519
C05099=1018.972,-58.966,-99.253,165.917,52.993,159.519
C05100=1018.977,-58.717,-99.264,165.920,52.988,159.518
C05101=1018.982,-58.467,-99.275,165.923,52.983,159.518
C05102=1018.988,-58.217,-99.285,165.926,52.978,159.518
C05103=1018.993,-57.967,-99.296,165.929,52.973,159.517
C05104=1018.999,-57.718,-99.307,165.932,52.967,159.517
C05105=1019.005,-57.468,-99.318,165.935,52.962,159.517
C05106=1019.010,-57.218,-99.328,165.938,52.957,159.516
C05107=1019.016,-56.969,-99.339,165.941,52.952,159.516
C05108=1019.022,-56.719,-99.350,165.943,52.947,159.515
C05109=1019.028,-56.470,-99.361,165.946,52.941,159.515
C05110=1019.033,-56.220,-99.371,165.949,52.936,159.515
C05111=1019.038,-55.970,-99.382,165.953,52.931,159.515
C05112=1019.044,-55.720,-99.393,165.956,52.926,159.514
C05113=1019.050,-55.471,-99.404,165.959,52.920,159.514
C05114=1019.055,-55.221,-99.414,165.962,52.915,159.513
C05115=1019.061,-54.971,-99.425,165.964,52.910,159.513
///RCONF 1,0,0,0,0,0,0,0,0,0,0,0,0,0,0,0,0,0,0,0,0,0,0,0
C05116=1019.066,-54.722,-99.436,165.967,52.904,159.513
C05117=1019.073,-54.471,-99.447,165.970,52.900,159.512
C05118=1019.079,-54.222,-99.458,165.973,52.894,159.512
C05119=1019.084,-53.972,-99.468,165.976,52.889,159.512
C05120=1019.090,-53.694,-99.481,165.979,52.883,159.511
C05121=1019.096,-53.416,-99.493,165.983,52.877,159.511
C05122=1019.102,-53.138,-99.505,165.986,52.872,159.511
C05123=1019.109,-52.859,-99.518,165.990,52.865,159.510
C05124=1019.115,-52.609,-99.528,165.992,52.860,159.510
C05125=1019.120,-52.360,-99.539,165.995,52.855,159.509
C05126=1019.126,-52.110,-99.549,165.998,52.849,159.509
C05127=1019.132,-51.861,-99.560,166.001,52.844,159.508
C05128=1019.138,-51.611,-99.571,166.004,52.839,159.508
C05129=1019.143,-51.361,-99.583,166.007,52.834,159.508
C05130=1019.149,-51.111,-99.594,166.010,52.829,159.508
C05131=1019.155,-50.862,-99.605,166.013,52.823,159.507
C05132=1019.160,-50.612,-99.616,166.015,52.818,159.507
C05133=1019.165,-50.363,-99.627,166.019,52.814,159.507
C05134=1019.170,-50.113,-99.639,166.022,52.808,159.506
C05135=1019.176,-49.863,-99.650,166.024,52.803,159.506
C05136=1019.182,-49.613,-99.661,166.027,52.798,159.505
C05137=1019.188,-49.364,-99.673,166.030,52.793,159.505
C05138=1019.193,-49.114,-99.684,166.033,52.788,159.505
C05139=1019.198,-48.865,-99.695,166.036,52.783,159.504
C05140=1019.203,-48.615,-99.707,166.039,52.778,159.504
C05141=1019.210,-48.365,-99.718,166.042,52.773,159.504
C05142=1019.215,-48.115,-99.730,166.045,52.768,159.504
C05143=1019.221,-47.865,-99.740,166.047,52.763,159.503
C05144=1019.226,-47.616,-99.753,166.050,52.758,159.503
C05145=1019.232,-47.367,-99.763,166.054,52.753,159.502
C05146=1019.237,-47.116,-99.775,166.057,52.748,159.502
C05147=1019.243,-46.867,-99.786,166.059,52.743,159.502
C05148=1019.248,-46.617,-99.798,166.063,52.738,159.501
C05149=1019.254,-46.368,-99.809,166.066,52.733,159.501
C05150=1019.259,-46.118,-99.821,166.068,52.727,159.501
C05151=1019.265,-45.868,-99.832,166.071,52.722,159.500
C05152=1019.270,-45.618,-99.843,166.074,52.717,159.500
C05153=1019.276,-45.369,-99.855,166.077,52.712,159.500
C05154=1019.281,-45.120,-99.866,166.080,52.707,159.499
C05155=1019.288,-44.869,-99.878,166.082,52.702,159.499
C05156=1019.293,-44.620,-99.889,166.086,52.697,159.499
C05157=1019.298,-44.370,-99.901,166.089,52.692,159.498
C05158=1019.304,-44.120,-99.913,166.092,52.686,159.498
C05159=1019.309,-43.870,-99.924,166.094,52.681,159.497
C05160=1019.315,-43.621,-99.936,166.097,52.677,159.497
C05161=1019.320,-43.372,-99.947,166.100,52.671,159.497
C05162=1019.327,-43.121,-99.958,166.103,52.666,159.496
C05163=1019.332,-42.872,-99.971,166.105,52.661,159.496
C05164=1019.338,-42.623,-99.981,166.108,52.656,159.496
C05165=1019.343,-42.372,-99.993,166.112,52.651,159.495
C05166=1019.349,-42.123,-100.005,166.115,52.646,159.495
C05167=1019.354,-41.874,-100.016,166.117,52.641,159.494
C05168=1019.361,-41.623,-100.028,166.120,52.635,159.494
C05169=1019.366,-41.374,-100.040,166.123,52.630,159.494
C05170=1019.372,-41.125,-100.051,166.127,52.625,159.494
C05171=1019.377,-40.874,-100.063,166.130,52.620,159.493
C05172=1019.383,-40.625,-100.075,166.132,52.615,159.493
C05173=1019.388,-40.376,-100.086,166.135,52.609,159.492
C05174=1019.394,-40.126,-100.098,166.138,52.604,159.492
C05175=1019.400,-39.876,-100.109,166.141,52.599,159.492
C05176=1019.405,-39.627,-100.121,166.143,52.594,159.491
C05177=1019.412,-39.377,-100.132,166.146,52.589,159.491
C05178=1019.417,-39.127,-100.144,166.149,52.584,159.490
C05179=1019.423,-38.877,-100.156,166.153,52.578,159.490
C05180=1019.428,-38.628,-100.169,166.155,52.573,159.490
C05181=1019.434,-38.379,-100.180,166.158,52.569,159.489
C05182=1019.440,-38.129,-100.192,166.161,52.563,159.489
C05183=1019.445,-37.879,-100.204,166.163,52.558,159.488
C05184=1019.451,-37.600,-100.217,166.167,52.553,159.488
C05185=1019.457,-37.323,-100.230,166.170,52.547,159.488
C05186=1019.463,-37.045,-100.243,166.173,52.541,159.487
C05187=1019.470,-36.767,-100.257,166.176,52.536,159.487
C05188=1019.475,-36.518,-100.269,166.179,52.530,159.487
C05189=1019.481,-36.268,-100.281,166.183,52.526,159.486
C05190=1019.486,-36.018,-100.293,166.185,52.521,159.486
C05191=1019.491,-35.769,-100.305,166.188,52.516,159.485
C05192=1019.498,-35.519,-100.317,166.191,52.510,159.485
C05193=1019.503,-35.269,-100.328,166.194,52.506,159.485
C05194=1019.509,-35.020,-100.341,166.196,52.501,159.484
C05195=1019.514,-34.770,-100.353,166.199,52.495,159.484
C05196=1019.520,-34.520,-100.365,166.202,52.490,159.484
C05197=1019.525,-34.271,-100.377,166.204,52.485,159.483
C05198=1019.532,-34.021,-100.389,166.208,52.480,159.483
C05199=1019.537,-33.771,-100.401,166.211,52.475,159.483
C05200=1019.543,-33.521,-100.413,166.214,52.470,159.482
C05201=1019.548,-33.272,-100.425,166.216,52.465,159.482
C05202=1019.554,-33.022,-100.437,166.219,52.459,159.481
C05203=1019.559,-32.773,-100.449,166.222,52.454,159.481
C05204=1019.566,-32.523,-100.461,166.226,52.449,159.481
C05205=1019.571,-32.274,-100.474,166.228,52.444,159.480
C05206=1019.576,-32.023,-100.485,166.231,52.439,159.480
C05207=1019.582,-31.774,-100.498,166.234,52.434,159.479
C05208=1019.588,-31.524,-100.510,166.237,52.428,159.479
C05209=1019.593,-31.275,-100.522,166.239,52.423,159.479
C05210=1019.600,-31.026,-100.534,166.242,52.418,159.478
C05211=1019.605,-30.776,-100.546,166.245,52.413,159.478
C05212=1019.611,-30.526,-100.558,166.247,52.408,159.477
C05213=1019.616,-30.277,-100.571,166.251,52.403,159.477
C05214=1019.622,-30.027,-100.583,166.254,52.398,159.477
C05215=1019.628,-29.777,-100.596,166.257,52.392,159.476
C05216=1019.633,-29.527,-100.606,166.260,52.387,159.476
C05217=1019.639,-29.278,-100.619,166.262,52.382,159.475
C05218=1019.645,-29.028,-100.631,166.265,52.377,159.475
C05219=1019.651,-28.778,-100.644,166.268,52.371,159.475
C05220=1019.656,-28.529,-100.656,166.271,52.366,159.474
C05221=1019.662,-28.279,-100.669,166.273,52.361,159.474
C05222=1019.668,-28.030,-100.680,166.276,52.356,159.473
C05223=1019.673,-27.780,-100.692,166.279,52.350,159.473
C05224=1019.679,-27.530,-100.705,166.282,52.345,159.473
C05225=1019.685,-27.281,-100.717,166.284,52.340,159.472
C05226=1019.691,-27.031,-100.729,166.288,52.335,159.472
C05227=1019.696,-26.781,-100.742,166.291,52.330,159.471
C05228=1019.701,-26.532,-100.755,166.293,52.325,159.471
C05229=1019.707,-26.282,-100.767,166.296,52.320,159.471
C05230=1019.713,-26.032,-100.780,166.299,52.314,159.470
C05231=1019.718,-25.783,-100.792,166.302,52.310,159.470
C05232=1019.724,-25.533,-100.804,166.305,52.305,159.469
C05233=1019.730,-25.283,-100.817,166.308,52.300,159.469
C05234=1019.736,-25.034,-100.830,166.310,52.295,159.469
C05235=1019.741,-24.784,-100.843,166.313,52.289,159.468
C05236=1019.746,-24.535,-100.855,166.316,52.284,159.468
C05237=1019.752,-24.285,-100.868,166.318,52.279,159.467
C05238=1019.758,-24.035,-100.880,166.322,52.274,159.467
C05239=1019.763,-23.786,-100.893,166.325,52.269,159.467
C05240=1019.769,-23.536,-100.905,166.327,52.264,159.466
C05241=1019.775,-23.286,-100.918,166.330,52.259,159.466
C05242=1019.780,-23.037,-100.930,166.333,52.253,159.465
C05243=1019.785,-22.787,-100.943,166.335,52.248,159.465
C05244=1019.792,-22.538,-100.956,166.338,52.243,159.465
C05245=1019.798,-22.288,-100.969,166.341,52.238,159.464
C05246=1019.803,-22.039,-100.981,166.344,52.232,159.464
C05247=1019.809,-21.789,-100.994,166.347,52.228,159.463
C05248=1019.815,-21.510,-101.008,166.351,52.222,159.463
C05249=1019.821,-21.231,-101.022,166.353,52.216,159.462
C05250=1019.828,-20.953,-101.036,166.356,52.211,159.462
C05251=1019.835,-20.674,-101.051,166.359,52.205,159.461
C05252=1019.840,-20.424,-101.063,166.362,52.199,159.461
C05253=1019.846,-20.175,-101.075,166.366,52.195,159.461
C05254=1019.852,-19.925,-101.088,166.368,52.190,159.460
C05255=1019.857,-19.675,-101.102,166.371,52.184,159.460
C05256=1019.862,-19.426,-101.114,166.374,52.179,159.459
C05257=1019.868,-19.176,-101.126,166.377,52.174,159.459
C05258=1019.874,-18.926,-101.139,166.379,52.169,159.459
C05259=1019.880,-18.676,-101.152,166.382,52.163,159.458
C05260=1019.886,-18.428,-101.164,166.385,52.158,159.458
C05261=1019.892,-18.178,-101.177,166.387,52.153,159.457
C05262=1019.897,-17.928,-101.190,166.390,52.148,159.457
C05263=1019.903,-17.678,-101.203,166.393,52.142,159.456
C05264=1019.908,-17.429,-101.216,166.396,52.137,159.456
C05265=1019.914,-17.179,-101.228,166.398,52.132,159.455
C05266=1019.920,-16.929,-101.241,166.401,52.126,159.455
C05267=1019.926,-16.680,-101.254,166.404,52.121,159.455
C05268=1019.932,-16.430,-101.267,166.407,52.116,159.454
C05269=1019.937,-16.180,-101.280,166.410,52.111,159.454
C05270=1019.943,-15.932,-101.293,166.413,52.105,159.453
C05271=1019.949,-15.682,-101.305,166.416,52.100,159.453
C05272=1019.954,-15.432,-101.319,166.418,52.095,159.452
C05273=1019.960,-15.182,-101.332,166.421,52.090,159.452
C05274=1019.966,-14.932,-101.344,166.424,52.085,159.452
C05275=1019.971,-14.683,-101.358,166.426,52.080,159.451
C05276=1019.977,-14.434,-101.370,166.430,52.075,159.451
C05277=1019.983,-14.184,-101.384,166.433,52.070,159.450
C05278=1019.988,-13.934,-101.397,166.435,52.065,159.450
C05279=1019.995,-13.685,-101.410,166.438,52.060,159.450
C05280=1020.000,-13.435,-101.423,166.441,52.054,159.449
C05281=1020.006,-13.185,-101.436,166.443,52.049,159.449
C05282=1020.011,-12.936,-101.449,166.446,52.044,159.448
C05283=1020.017,-12.687,-101.462,166.449,52.039,159.448
C05284=1020.022,-12.437,-101.476,166.451,52.034,159.447
C05285=1020.028,-12.187,-101.489,166.454,52.028,159.447
C05286=1020.034,-11.938,-101.502,166.458,52.023,159.447
C05287=1020.040,-11.688,-101.515,166.460,52.018,159.446
C05288=1020.046,-11.438,-101.528,166.463,52.013,159.446
C05289=1020.051,-11.188,-101.542,166.466,52.008,159.445
C05290=1020.057,-10.940,-101.555,166.468,52.003,159.445
C05291=1020.062,-10.689,-101.568,166.471,51.997,159.444
C05292=1020.068,-10.440,-101.581,166.474,51.992,159.444
C05293=1020.074,-10.191,-101.594,166.476,51.987,159.443
C05294=1020.079,-9.941,-101.607,166.479,51.982,159.443
C05295=1020.086,-9.691,-101.621,166.482,51.977,159.443
C05296=1020.091,-9.441,-101.634,166.485,51.972,159.442
C05297=1020.097,-9.192,-101.647,166.488,51.966,159.442
C05298=1020.102,-8.942,-101.661,166.491,51.961,159.441
C05299=1020.108,-8.693,-101.673,166.493,51.956,159.441
C05300=1020.115,-8.443,-101.687,166.496,51.951,159.440
C05301=1020.120,-8.194,-101.701,166.499,51.946,159.440
C05302=1020.126,-7.944,-101.713,166.501,51.941,159.439
C05303=1020.131,-7.694,-101.727,166.504,51.935,159.439
C05304=1020.138,-7.445,-101.740,166.507,51.929,159.438
C05305=1020.143,-7.195,-101.753,166.510,51.924,159.438
C05306=1020.149,-6.946,-101.767,166.512,51.919,159.437
C05307=1020.155,-6.697,-101.780,166.515,51.914,159.437
C05308=1020.160,-6.447,-101.793,166.518,51.909,159.437
C05309=1020.166,-6.198,-101.806,166.520,51.904,159.436
C05310=1020.171,-5.948,-101.820,166.524,51.898,159.436
C05311=1020.178,-5.699,-101.833,166.527,51.893,159.435
C05312=1020.184,-5.417,-101.848,166.529,51.887,159.435
C05313=1020.191,-5.137,-101.864,166.532,51.881,159.434
C05314=1020.198,-4.856,-101.878,166.536,51.875,159.434
C05315=1020.204,-4.575,-101.893,166.539,51.869,159.433
C05316=1020.210,-4.326,-101.906,166.542,51.864,159.433
C05317=1020.215,-4.077,-101.920,166.544,51.859,159.432
C05318=1020.221,-3.827,-101.934,166.547,51.853,159.432
C05319=1020.226,-3.577,-101.948,166.549,51.848,159.431
C05320=1020.232,-3.328,-101.962,166.552,51.843,159.431
C05321=1020.238,-3.079,-101.975,166.555,51.838,159.430
C05322=1020.244,-2.829,-101.989,166.557,51.833,159.430
C05323=1020.249,-2.579,-102.003,166.561,51.828,159.430
C05324=1020.254,-2.329,-102.016,166.563,51.824,159.429
C05325=1020.260,-2.080,-102.030,166.566,51.818,159.429
C05326=1020.266,-1.830,-102.043,166.569,51.813,159.428
C05327=1020.271,-1.581,-102.057,166.571,51.808,159.428
C05328=1020.277,-1.331,-102.071,166.574,51.803,159.427
C05329=1020.283,-1.081,-102.085,166.577,51.798,159.427
C05330=1020.288,-0.831,-102.099,166.580,51.793,159.426
C05331=1020.295,-0.582,-102.112,166.583,51.787,159.426
C05332=1020.300,-0.333,-102.126,166.585,51.782,159.426
C05333=1020.306,-0.083,-102.140,166.588,51.777,159.425
C05334=1020.311,0.167,-102.154,166.590,51.772,159.425
C05335=1020.317,0.416,-102.168,166.593,51.767,159.424
C05336=1020.322,0.665,-102.182,166.596,51.762,159.424
C05337=1020.329,0.914,-102.195,166.598,51.756,159.423
C05338=1020.334,1.164,-102.209,166.601,51.751,159.423
C05339=1020.339,1.413,-102.223,166.603,51.746,159.422
C05340=1020.345,1.663,-102.237,166.606,51.741,159.422
C05341=1020.351,1.913,-102.251,166.610,51.735,159.421
C05342=1020.357,2.163,-102.264,166.612,51.731,159.421
C05343=1020.363,2.412,-102.278,166.615,51.725,159.420
C05344=1020.368,2.662,-102.292,166.618,51.720,159.420
C05345=1020.374,2.911,-102.306,166.620,51.715,159.419
C05346=1020.379,3.161,-102.320,166.623,51.710,159.419
C05347=1020.385,3.410,-102.334,166.625,51.705,159.419
C05348=1020.392,3.660,-102.348,166.628,51.700,159.418
C05349=1020.397,3.909,-102.362,166.631,51.694,159.418
C05350=1020.403,4.159,-102.376,166.633,51.689,159.417
C05351=1020.408,4.409,-102.390,166.636,51.684,159.417
C05352=1020.414,4.658,-102.404,166.640,51.678,159.416
C05353=1020.420,4.907,-102.417,166.642,51.673,159.416
C05354=1020.426,5.158,-102.431,166.645,51.668,159.415
C05355=1020.432,5.407,-102.446,166.648,51.663,159.415
C05356=1020.437,5.656,-102.460,166.650,51.657,159.414
C05357=1020.443,5.906,-102.473,166.653,51.652,159.414
C05358=1020.448,6.155,-102.487,166.655,51.647,159.413
C05359=1020.455,6.405,-102.501,166.658,51.642,159.413
C05360=1020.461,6.654,-102.516,166.661,51.637,159.412
C05361=1020.466,6.904,-102.529,166.663,51.631,159.412
C05362=1020.472,7.153,-102.543,166.666,51.626,159.411
C05363=1020.477,7.403,-102.557,166.669,51.621,159.411
C05364=1020.483,7.653,-102.571,166.671,51.616,159.410
C05365=1020.490,7.902,-102.585,166.674,51.610,159.410
C05366=1020.495,8.152,-102.599,166.677,51.605,159.409
C05367=1020.501,8.401,-102.613,166.679,51.600,159.409
C05368=1020.507,8.651,-102.627,166.682,51.594,159.408
C05369=1020.513,8.900,-102.642,166.686,51.589,159.408
C05370=1020.518,9.150,-102.656,166.687,51.584,159.407
C05371=1020.524,9.399,-102.670,166.690,51.578,159.407
C05372=1020.531,9.649,-102.684,166.694,51.573,159.406
C05373=1020.536,9.898,-102.698,166.696,51.568,159.406
C05374=1020.542,10.148,-102.712,166.698,51.562,159.405
C05375=1020.547,10.398,-102.726,166.702,51.557,159.405
C05376=1020.554,10.680,-102.742,166.704,51.551,159.404
C05377=1020.561,10.962,-102.758,166.707,51.545,159.404
C05378=1020.568,11.245,-102.774,166.711,51.539,159.403
